  MoveL 769 to (-578.4, 1200, 50) mm, rotated rx -180 ry 0 rz 90 deg; joints [-4.57, -97.989, 142.035, 22.266, 7.604, -25.643]
  MoveL 770 to (-578.4, 1200, -0.5) mm, rotated rx -180 ry 0 rz 90 deg; joints [-4.57, -94.77, 142.936, 44.544, 4.099, -48.025]
  MoveL 771 to (-578.4, 1200, 50) mm, rotated rx -180 ry 0 rz 90 deg; joints [-4.57, -97.989, 142.035, 22.266, 7.604, -25.643]
  MoveL 772 to (-578.4, 1250, 50) mm, rotated rx -180 ry 0 rz 90 deg; joints [-4.804, -101.028, 144.386, 21.399, 8.305, -24.931]
  MoveL 773 to (-578.4, 1250, -0.5) mm, rotated rx 180 ry 0 rz 90 deg; joints [-4.804, -97.638, 145.343, 41.717, 4.543, -45.364]
  MoveL 774 to (-578.4, 1250, 50) mm, rotated rx -180 ry 0 rz 90 deg; joints [-4.804, -101.028, 144.386, 21.399, 8.305, -24.931]
  MoveL 775 to (-578.4, 1300, 50) mm, rotated rx -180 ry 0 rz 90 deg; joints [-5.063, -104.304, 146.692, 20.148, 9.28, -23.844]
  MoveL 776 to (-578.4, 1300, -0.5) mm, rotated rx 180 ry 0 rz 90 deg; joints [-5.063, -100.735, 147.713, 37.677, 5.214, -41.502]
  MoveL 777 to (-578.4, 1300, 50) mm, rotated rx -180 ry 0 rz 90 deg; joints [-5.063, -104.304, 146.692, 20.148, 9.28, -23.844]
  MoveL 778 to (-578.4, 1350, 50) mm, rotated rx 180 ry 0 rz 90 deg; joints [-5.353, -107.868, 148.948, 18.637, 10.585, -22.506]
  MoveL 779 to (-578.4, 1350, -0.5) mm, rotated rx 180 ry 0 rz 90 deg; joints [-5.353, -104.114, 150.044, 33.013, 6.186, -37.025]
  MoveL 780 to (-578.4, 1350, 50) mm, rotated rx 180 ry 0 rz 90 deg; joints [-5.353, -107.868, 148.948, 18.637, 10.585, -22.506]
  MoveL 781 to (-578.4, 1400, 50) mm, rotated rx 180 ry 0 rz 90 deg; joints [-5.676, -111.783, 151.148, 16.997, 12.295, -21.046]
  MoveL 782 to (-578.4, 1400, -0.5) mm, rotated rx 180 ry 0 rz 90 deg; joints [-5.676, -107.847, 152.329, 28.286, 7.548, -32.495]
  MoveL 783 to (-578.4, 1400, 50) mm, rotated rx 180 ry 0 rz 90 deg; joints [-5.676, -111.783, 151.148, 16.997, 12.295, -21.046]
  MoveL 784 to (-578.4, 1450, 50) mm, rotated rx -180 ry 0 rz 90 deg; joints [-6.042, -116.128, 153.28, 15.341, 14.499, -19.577]
  MoveL 785 to (-578.4, 1450, -0.5) mm, rotated rx 180 ry 0 rz 90 deg; joints [-6.042, -112.023, 154.561, 23.895, 9.412, -28.311]
  MoveL 786 to (-578.4, 1450, 50) mm, rotated rx -180 ry 0 rz 90 deg; joints [-6.042, -116.128, 153.28, 15.341, 14.499, -19.577]
  MoveL 787 to (-514.2, 300, 50) mm, rotated rx 180 ry 0 rz 90 deg; joints [-4.34, -58.339, 92.264, 9.183, 17.364, -12.147]
  MoveL 788 to (-514.2, 300, -0.5) mm, rotated rx -180 ry 0 rz 90 deg; joints [-4.34, -56.823, 92.789, 10.363, 15.353, -13.377]
  MoveL 789 to (-514.2, 300, 50) mm, rotated rx 180 ry 0 rz 90 deg; joints [-4.34, -58.339, 92.264, 9.183, 17.364, -12.147]
  MoveL 790 to (-514.2, 650, 50) mm, rotated rx -180 ry 0 rz 90 deg; joints [-5.302, -72.243, 113.368, 18.554, 10.531, -22.388]
  MoveL 791 to (-514.2, 650, -0.5) mm, rotated rx 180 ry 0 rz 90 deg; joints [-5.302, -70.292, 113.949, 24.154, 8.171, -28.062]
  MoveL 792 to (-514.2, 650, 50) mm, rotated rx -180 ry 0 rz 90 deg; joints [-5.302, -72.243, 113.368, 18.554, 10.531, -22.388]
  MoveL 793 to (-476, 230, 50) mm, rotated rx -180 ry 0 rz 90 deg; joints [-5.28, -55.357, 87.377, 10.054, 19.374, -13.603]
  MoveL 794 to (-476, 230, -0.5) mm, rotated rx 180 ry 0 rz 90 deg; joints [-5.28, -53.915, 87.901, 11.14, 17.442, -14.748]
  MoveL 795 to (-476, 230, 50) mm, rotated rx -180 ry 0 rz 90 deg; joints [-5.28, -55.357, 87.377, 10.054, 19.374, -13.603]
  MoveL 796 to (-514.2, 230, 50) mm, rotated rx 180 ry 0 rz 90 deg; joints [-4.188, -55.487, 87.593, 8.057, 19.144, -10.874]
  MoveL 797 to (-514.2, 230, -0.5) mm, rotated rx -180 ry 0 rz 90 deg; joints [-4.188, -54.042, 88.116, 8.943, 17.198, -11.807]
  MoveL 798 to (-514.2, 230, 50) mm, rotated rx 180 ry 0 rz 90 deg; joints [-4.188, -55.487, 87.593, 8.057, 19.144, -10.874]
  MoveL 799 to (-552.4, 230, 50) mm, rotated rx -180 ry 0 rz 90 deg; joints [-3.094, -55.587, 87.758, 5.998, 18.966, -8.08]
  MoveL 800 to (-552.4, 230, -0.5) mm, rotated rx -180 ry 0 rz 90 deg; joints [-3.094, -54.14, 88.282, 6.668, 17.007, -8.784]
  MoveL 801 to (-552.4, 230, 50) mm, rotated rx -180 ry 0 rz 90 deg; joints [-3.094, -55.587, 87.758, 5.998, 18.966, -8.08]
  MoveL 802 to (-655, 50, 50) mm, rotated rx 180 ry 0 rz 90 deg; joints [-0.132, -48.006, 74.913, 0.203, 24.093, -0.288]
  MoveL 803 to (-655, 50, -0.5) mm, rotated rx 180 ry 0 rz 90 deg; joints [-0.132, -46.724, 75.45, 0.219, 22.275, -0.305]
  MoveL 804 to (-655, 50, 50) mm, rotated rx 180 ry 0 rz 90 deg; joints [-0.132, -48.006, 74.913, 0.203, 24.093, -0.288]
  MoveL 805 to (-655, 100, 50) mm, rotated rx 180 ry 0 rz 90 deg; joints [-0.135, -50.213, 78.713, 0.222, 22.501, -0.31]
  MoveL 806 to (-655, 100, -0.5) mm, rotated rx 180 ry 0 rz 90 deg; joints [-0.135, -48.886, 79.243, 0.241, 20.644, -0.331]
  MoveL 807 to (-655, 100, 50) mm, rotated rx 180 ry 0 rz 90 deg; joints [-0.135, -50.213, 78.713, 0.222, 22.501, -0.31]
  MoveL 808 to (-655, 150, 50) mm, rotated rx 180 ry 0 rz 90 deg; joints [-0.138, -52.362, 82.367, 0.243, 20.996, -0.334]
  MoveL 809 to (-655, 150, -0.5) mm, rotated rx -180 ry 0 rz 90 deg; joints [-0.138, -50.989, 82.893, 0.266, 19.097, -0.359]
  MoveL 810 to (-655, 150, 50) mm, rotated rx 180 ry 0 rz 90 deg; joints [-0.138, -52.362, 82.367, 0.243, 20.996, -0.334]
  MoveL 811 to (-655, 200, 50) mm, rotated rx 180 ry 0 rz 90 deg; joints [-0.142, -54.464, 85.894, 0.266, 19.57, -0.361]
  MoveL 812 to (-655, 200, -0.5) mm, rotated rx 180 ry 0 rz 90 deg; joints [-0.142, -53.043, 86.418, 0.295, 17.626, -0.391]
  MoveL 813 to (-655, 200, 50) mm, rotated rx 180 ry 0 rz 90 deg; joints [-0.142, -54.464, 85.894, 0.266, 19.57, -0.361]
  MoveL 814 to (-655, 250, 50) mm, rotated rx 180 ry 0 rz 90 deg; joints [-0.145, -56.528, 89.31, 0.293, 18.219, -0.391]
  MoveL 815 to (-655, 250, -0.5) mm, rotated rx 180 ry 0 rz 90 deg; joints [-0.145, -55.058, 89.833, 0.327, 16.225, -0.427]
  MoveL 816 to (-655, 250, 50) mm, rotated rx 180 ry 0 rz 90 deg; joints [-0.145, -56.528, 89.31, 0.293, 18.219, -0.391]
  MoveL 817 to (-655, 300, 50) mm, rotated rx -180 ry 0 rz 90 deg; joints [-0.149, -58.562, 92.626, 0.322, 16.937, -0.424]
  MoveL 818 to (-655, 300, -0.5) mm, rotated rx 180 ry 0 rz 90 deg; joints [-0.149, -57.041, 93.151, 0.365, 14.89, -0.469]
  MoveL 819 to (-655, 300, 50) mm, rotated rx -180 ry 0 rz 90 deg; joints [-0.149, -58.562, 92.626, 0.322, 16.937, -0.424]
  MoveL 820 to (-655, 350, 50) mm, rotated rx 180 ry 0 rz 90 deg; joints [-0.153, -60.573, 95.852, 0.356, 15.721, -0.461]
  MoveL 821 to (-655, 350, -0.5) mm, rotated rx -180 ry 0 rz 90 deg; joints [-0.153, -58.998, 96.381, 0.409, 13.618, -0.517]
  MoveL 822 to (-655, 350, 50) mm, rotated rx 180 ry 0 rz 90 deg; joints [-0.153, -60.573, 95.852, 0.356, 15.721, -0.461]
  MoveL 823 to (-655, 400, 50) mm, rotated rx -180 ry 0 rz 90 deg; joints [-0.157, -62.568, 98.998, 0.394, 14.57, -0.503]
  MoveL 824 to (-655, 400, -0.5) mm, rotated rx 180 ry 0 rz 90 deg; joints [-0.157, -60.937, 99.532, 0.461, 12.406, -0.572]
  MoveL 825 to (-655, 400, 50) mm, rotated rx -180 ry 0 rz 90 deg; joints [-0.157, -62.568, 98.998, 0.394, 14.57, -0.503]
  MoveL 826 to (-655, 450, 50) mm, rotated rx -180 ry 0 rz 90 deg; joints [-0.162, -64.553, 102.071, 0.437, 13.482, -0.55]
  MoveL 827 to (-655, 450, -0.5) mm, rotated rx 180 ry 0 rz 90 deg; joints [-0.162, -62.863, 102.612, 0.522, 11.252, -0.637]
  MoveL 828 to (-655, 450, 50) mm, rotated rx -180 ry 0 rz 90 deg; joints [-0.162, -64.553, 102.071, 0.437, 13.482, -0.55]
  MoveL 829 to (-655, 500, 50) mm, rotated rx -180 ry 0 rz 90 deg; joints [-0.166, -66.534, 105.078, 0.486, 12.457, -0.604]
  MoveL 830 to (-655, 500, -0.5) mm, rotated rx -180 ry 0 rz 90 deg; joints [-0.166, -64.782, 105.626, 0.594, 10.157, -0.714]
  MoveL 831 to (-655, 500, 50) mm, rotated rx -180 ry 0 rz 90 deg; joints [-0.166, -66.534, 105.078, 0.486, 12.457, -0.604]
  MoveL 832 to (-655, 550, 50) mm, rotated rx 180 ry 0 rz 90 deg; joints [-0.171, -68.517, 108.023, 0.541, 11.495, -0.664]
  MoveL 833 to (-655, 550, -0.5) mm, rotated rx -180 ry 0 rz 90 deg; joints [-0.171, -66.7, 108.581, 0.681, 9.12, -0.805]
  MoveL 834 to (-655, 550, 50) mm, rotated rx 180 ry 0 rz 90 deg; joints [-0.171, -68.517, 108.023, 0.541, 11.495, -0.664]
  MoveL 835 to (-655, 600, 50) mm, rotated rx -180 ry 0 rz 90 deg; joints [-0.177, -70.508, 110.911, 0.605, 10.598, -0.732]
  MoveL 836 to (-655, 600, -0.5) mm, rotated rx -180 ry 0 rz 90 deg; joints [-0.177, -68.622, 111.481, 0.785, 8.142, -0.915]
  MoveL 837 to (-655, 600, 50) mm, rotated rx -180 ry 0 rz 90 deg; joints [-0.177, -70.508, 110.911, 0.605, 10.598, -0.732]
  MoveL 838 to (-655, 650, 50) mm, rotated rx -180 ry 0 rz 90 deg; joints [-0.182, -72.515, 113.748, 0.676, 9.768, -0.808]
  MoveL 839 to (-655, 650, -0.5) mm, rotated rx 180 ry 0 rz 90 deg; joints [-0.182, -70.554, 114.33, 0.913, 7.225, -1.047]
  MoveL 840 to (-655, 650, 50) mm, rotated rx -180 ry 0 rz 90 deg; joints [-0.182, -72.515, 113.748, 0.676, 9.768, -0.808]
  MoveL 841 to (-655, 700, 50) mm, rotated rx 180 ry 0 rz 90 deg; joints [-0.188, -74.542, 116.535, 0.757, 9.008, -0.894]
  MoveL 842 to (-655, 700, -0.5) mm, rotated rx 180 ry 0 rz 90 deg; joints [-0.188, -72.503, 117.133, 1.068, 6.371, -1.208]
  MoveL 843 to (-655, 700, 50) mm, rotated rx 180 ry 0 rz 90 deg; joints [-0.188, -74.542, 116.535, 0.757, 9.008, -0.894]
  MoveL 844 to (-655, 750, 50) mm, rotated rx -180 ry 0 rz 90 deg; joints [-0.195, -76.598, 119.277, 0.847, 8.323, -0.989]
  MoveL 845 to (-655, 750, -0.5) mm, rotated rx 180 ry 0 rz 90 deg; joints [-0.195, -74.475, 119.891, 1.26, 5.585, -1.405]
  MoveL 846 to (-655, 750, 50) mm, rotated rx -180 ry 0 rz 90 deg; joints [-0.195, -76.598, 119.277, 0.847, 8.323, -0.989]
  MoveL 847 to (-655, 800, 50) mm, rotated rx -180 ry 0 rz 90 deg; joints [-0.202, -78.691, 121.976, 0.945, 7.717, -1.093]
  MoveL 848 to (-655, 800, -0.5) mm, rotated rx 180 ry 0 rz 90 deg; joints [-0.202, -76.477, 122.609, 1.495, 4.87, -1.646]
  MoveL 849 to (-655, 800, 50) mm, rotated rx -180 ry 0 rz 90 deg; joints [-0.202, -78.691, 121.976, 0.945, 7.717, -1.093]
  MoveL 850 to (-655, 850, 50) mm, rotated rx 180 ry 0 rz 90 deg; joints [-0.209, -80.83, 124.634, 1.05, 7.198, -1.204]
  MoveL 851 to (-655, 850, -0.5) mm, rotated rx -180 ry 0 rz 90 deg; joints [-0.209, -78.519, 125.288, 1.782, 4.233, -1.94]
  MoveL 852 to (-655, 850, 50) mm, rotated rx 180 ry 0 rz 90 deg; joints [-0.209, -80.83, 124.634, 1.05, 7.198, -1.204]
  MoveL 853 to (-655, 900, 50) mm, rotated rx 180 ry 0 rz 90 deg; joints [-0.217, -83.024, 127.252, 1.157, 6.773, -1.318]
  MoveL 854 to (-655, 900, -0.5) mm, rotated rx -180 ry 0 rz 90 deg; joints [-0.217, -80.609, 127.931, 2.127, 3.681, -2.291]
  MoveL 855 to (-655, 900, 50) mm, rotated rx 180 ry 0 rz 90 deg; joints [-0.217, -83.024, 127.252, 1.157, 6.773, -1.318]
  MoveL 856 to (-655, 950, 50) mm, rotated rx 180 ry 0 rz 90 deg; joints [-0.225, -85.286, 129.834, 1.262, 6.454, -1.429]
  MoveL 857 to (-655, 950, -0.5) mm, rotated rx 180 ry 0 rz 90 deg; joints [-0.225, -82.759, 130.54, 2.524, 3.223, -2.695]
  MoveL 858 to (-655, 950, 50) mm, rotated rx 180 ry 0 rz 90 deg; joints [-0.225, -85.286, 129.834, 1.262, 6.454, -1.429]
  MoveL 859 to (-655, 1000, 50) mm, rotated rx 180 ry 0 rz 90 deg; joints [-0.235, -87.628, 132.378, 1.356, 6.252, -1.53]
  MoveL 860 to (-655, 1000, -0.5) mm, rotated rx 180 ry 0 rz 90 deg; joints [-0.235, -84.981, 133.115, 2.95, 2.87, -3.129]
  MoveL 861 to (-655, 1000, 50) mm, rotated rx 180 ry 0 rz 90 deg; joints [-0.235, -87.628, 132.378, 1.356, 6.252, -1.53]
  MoveL 862 to (-655, 1050, 50) mm, rotated rx 180 ry 0 rz 90 deg; joints [-0.245, -90.068, 134.886, 1.429, 6.184, -1.611]
  MoveL 863 to (-655, 1050, -0.5) mm, rotated rx 180 ry 0 rz 90 deg; joints [-0.245, -87.291, 135.657, 3.347, 2.638, -3.534]
  MoveL 864 to (-655, 1050, 50) mm, rotated rx 180 ry 0 rz 90 deg; joints [-0.245, -90.068, 134.886, 1.429, 6.184, -1.611]
  MoveL 865 to (-655, 1100, 50) mm, rotated rx 180 ry 0 rz 90 deg; joints [-0.256, -92.624, 137.358, 1.473, 6.268, -1.663]
  MoveL 866 to (-655, 1100, -0.5) mm, rotated rx -180 ry 0 rz 90 deg; joints [-0.256, -89.706, 138.168, 3.626, 2.544, -3.821]
  MoveL 867 to (-655, 1100, 50) mm, rotated rx 180 ry 0 rz 90 deg; joints [-0.256, -92.624, 137.358, 1.473, 6.268, -1.663]
  MoveL 868 to (-655, 1150, 50) mm, rotated rx -180 ry 0 rz 90 deg; joints [-0.267, -95.319, 139.793, 1.481, 6.528, -1.679]
  MoveL 869 to (-655, 1150, -0.5) mm, rotated rx -180 ry 0 rz 90 deg; joints [-0.267, -92.25, 140.647, 3.7, 2.609, -3.904]
  MoveL 870 to (-655, 1150, 50) mm, rotated rx -180 ry 0 rz 90 deg; joints [-0.267, -95.319, 139.793, 1.481, 6.528, -1.679]
  MoveL 871 to (-655, 1200, 50) mm, rotated rx -180 ry 0 rz 90 deg; joints [-0.281, -98.18, 142.19, 1.45, 6.993, -1.658]
  MoveL 872 to (-655, 1200, -0.5) mm, rotated rx 180 ry 0 rz 90 deg; joints [-0.281, -94.951, 143.093, 3.537, 2.863, -3.751]
  MoveL 873 to (-655, 1200, 50) mm, rotated rx -180 ry 0 rz 90 deg; joints [-0.281, -98.18, 142.19, 1.45, 6.993, -1.658]
  MoveL 874 to (-655, 1250, 50) mm, rotated rx 180 ry 0 rz 90 deg; joints [-0.295, -101.244, 144.545, 1.386, 7.701, -1.603]
  MoveL 875 to (-655, 1250, -0.5) mm, rotated rx 180 ry 0 rz 90 deg; joints [-0.295, -97.842, 145.506, 3.187, 3.342, -3.411]
  MoveL 876 to (-655, 1250, 50) mm, rotated rx 180 ry 0 rz 90 deg; joints [-0.295, -101.244, 144.545, 1.386, 7.701, -1.603]
  MoveL 877 to (-783.4, 50, 50) mm, rotated rx 180 ry 0 rz 90 deg; joints [3.253, -47.849, 74.641, -4.972, 24.334, 7.062]
  MoveL 878 to (-783.4, 50, -0.5) mm, rotated rx 180 ry 0 rz 90 deg; joints [3.253, -46.571, 75.179, -5.349, 22.525, 7.473]
  MoveL 879 to (-783.4, 50, 50) mm, rotated rx 180 ry 0 rz 90 deg; joints [3.253, -47.849, 74.641, -4.972, 24.334, 7.062]
  MoveL 880 to (-783.4, 100, 50) mm, rotated rx 180 ry 0 rz 90 deg; joints [3.33, -50.057, 78.445, -5.424, 22.75, 7.593]
  MoveL 881 to (-783.4, 100, -0.5) mm, rotated rx -180 ry 0 rz 90 deg; joints [3.33, -48.733, 78.976, -5.88, 20.905, 8.084]
  MoveL 882 to (-783.4, 100, 50) mm, rotated rx 180 ry 0 rz 90 deg; joints [3.33, -50.057, 78.445, -5.424, 22.75, 7.593]
  MoveL 883 to (-783.4, 150, 50) mm, rotated rx 180 ry 0 rz 90 deg; joints [3.41, -52.206, 82.103, -5.926, 21.256, 8.177]
  MoveL 884 to (-783.4, 150, -0.5) mm, rotated rx 180 ry 0 rz 90 deg; joints [3.41, -50.837, 82.629, -6.48, 19.371, 8.767]
  MoveL 885 to (-783.4, 150, 50) mm, rotated rx 180 ry 0 rz 90 deg; joints [3.41, -52.206, 82.103, -5.926, 21.256, 8.177]
  MoveL 886 to (-783.4, 200, 50) mm, rotated rx -180 ry 0 rz 90 deg; joints [3.494, -54.308, 85.633, -6.488, 19.844, 8.822]
  MoveL 887 to (-783.4, 200, -0.5) mm, rotated rx -180 ry 0 rz 90 deg; joints [3.494, -52.89, 86.157, -7.162, 17.917, 9.535]
  MoveL 888 to (-783.4, 200, 50) mm, rotated rx -180 ry 0 rz 90 deg; joints [3.494, -54.308, 85.633, -6.488, 19.844, 8.822]
  MoveL 889 to (-783.4, 250, 50) mm, rotated rx 180 ry 0 rz 90 deg; joints [3.583, -56.37, 89.05, -7.116, 18.508, 9.537]
  MoveL 890 to (-783.4, 250, -0.5) mm, rotated rx -180 ry 0 rz 90 deg; joints [3.583, -54.904, 89.574, -7.942, 16.535, 10.403]
  MoveL 891 to (-783.4, 250, 50) mm, rotated rx 180 ry 0 rz 90 deg; joints [3.583, -56.37, 89.05, -7.116, 18.508, 9.537]
  MoveL 892 to (-783.4, 300, 50) mm, rotated rx 180 ry 0 rz 90 deg; joints [3.676, -58.402, 92.367, -7.822, 17.244, 10.332]
  MoveL 893 to (-783.4, 300, -0.5) mm, rotated rx -180 ry 0 rz 90 deg; joints [3.676, -56.885, 92.892, -8.838, 15.223, 11.391]
  MoveL 894 to (-783.4, 300, 50) mm, rotated rx 180 ry 0 rz 90 deg; joints [3.676, -58.402, 92.367, -7.822, 17.244, 10.332]
  MoveL 895 to (-783.4, 350, 50) mm, rotated rx 180 ry 0 rz 90 deg; joints [3.774, -60.41, 95.593, -8.616, 16.05, 11.219]
  MoveL 896 to (-783.4, 350, -0.5) mm, rotated rx 180 ry 0 rz 90 deg; joints [3.774, -58.84, 96.122, -9.873, 13.978, 12.52]
  MoveL 897 to (-783.4, 350, 50) mm, rotated rx 180 ry 0 rz 90 deg; joints [3.774, -60.41, 95.593, -8.616, 16.05, 11.219]
  MoveL 898 to (-783.4, 400, 50) mm, rotated rx 180 ry 0 rz 90 deg; joints [3.877, -62.402, 98.739, -9.51, 14.923, 12.21]
  MoveL 899 to (-783.4, 400, -0.5) mm, rotated rx 180 ry 0 rz 90 deg; joints [3.877, -60.776, 99.272, -11.074, 12.799, 13.82]
  MoveL 900 to (-783.4, 400, 50) mm, rotated rx 180 ry 0 rz 90 deg; joints [3.877, -62.402, 98.739, -9.51, 14.923, 12.21]
  MoveL 901 to (-783.4, 450, 50) mm, rotated rx 180 ry 0 rz 90 deg; joints [3.986, -64.383, 101.811, -10.519, 13.864, 13.319]
  MoveL 902 to (-783.4, 450, -0.5) mm, rotated rx 180 ry 0 rz 90 deg; joints [3.986, -62.698, 102.35, -12.474, 11.685, 15.323]
  MoveL 903 to (-783.4, 450, 50) mm, rotated rx 180 ry 0 rz 90 deg; joints [3.986, -64.383, 101.811, -10.519, 13.864, 13.319]
  MoveL 904 to (-783.4, 500, 50) mm, rotated rx -180 ry 0 rz 90 deg; joints [4.101, -66.359, 104.815, -11.656, 12.873, 14.56]
  MoveL 905 to (-783.4, 500, -0.5) mm, rotated rx -180 ry 0 rz 90 deg; joints [4.101, -64.613, 105.363, -14.114, 10.636, 17.071]
  MoveL 906 to (-783.4, 500, 50) mm, rotated rx -180 ry 0 rz 90 deg; joints [4.101, -66.359, 104.815, -11.656, 12.873, 14.56]
  MoveL 907 to (-783.4, 550, 50) mm, rotated rx 180 ry 0 rz 90 deg; joints [4.224, -68.337, 107.758, -12.935, 11.95, 15.949]
  MoveL 908 to (-783.4, 550, -0.5) mm, rotated rx 180 ry 0 rz 90 deg; joints [4.224, -66.525, 108.315, -16.041, 9.656, 19.11]
  MoveL 909 to (-783.4, 550, 50) mm, rotated rx 180 ry 0 rz 90 deg; joints [4.224, -68.337, 107.758, -12.935, 11.95, 15.949]
  MoveL 910 to (-783.4, 600, 50) mm, rotated rx 180 ry 0 rz 90 deg; joints [4.353, -70.321, 110.643, -14.369, 11.098, 17.497]
  MoveL 911 to (-783.4, 600, -0.5) mm, rotated rx 180 ry 0 rz 90 deg; joints [4.353, -68.441, 111.211, -18.308, 8.747, 21.495]
  MoveL 912 to (-783.4, 600, 50) mm, rotated rx 180 ry 0 rz 90 deg; joints [4.353, -70.321, 110.643, -14.369, 11.098, 17.497]
  MoveL 913 to (-783.4, 650, 50) mm, rotated rx -180 ry 0 rz 90 deg; joints [4.491, -72.32, 113.476, -15.967, 10.32, 19.215]
  MoveL 914 to (-783.4, 650, -0.5) mm, rotated rx 180 ry 0 rz 90 deg; joints [4.491, -70.367, 114.057, -20.973, 7.914, 24.283]
  MoveL 915 to (-783.4, 650, 50) mm, rotated rx -180 ry 0 rz 90 deg; joints [4.491, -72.32, 113.476, -15.967, 10.32, 19.215]
  MoveL 916 to (-783.4, 700, 50) mm, rotated rx 180 ry 0 rz 90 deg; joints [4.638, -74.339, 116.259, -17.729, 9.621, 21.103]
  MoveL 917 to (-783.4, 700, -0.5) mm, rotated rx -180 ry 0 rz 90 deg; joints [4.638, -72.307, 116.855, -24.09, 7.162, 27.531]
  MoveL 918 to (-783.4, 700, 50) mm, rotated rx 180 ry 0 rz 90 deg; joints [4.638, -74.339, 116.259, -17.729, 9.621, 21.103]
  MoveL 919 to (-783.4, 750, 50) mm, rotated rx -180 ry 0 rz 90 deg; joints [4.795, -76.385, 118.996, -19.645, 9.003, 23.152]
  MoveL 920 to (-783.4, 750, -0.5) mm, rotated rx 180 ry 0 rz 90 deg; joints [4.795, -74.27, 119.609, -27.698, 6.499, 31.277]
  MoveL 921 to (-783.4, 750, 50) mm, rotated rx -180 ry 0 rz 90 deg; joints [4.795, -76.385, 118.996, -19.645, 9.003, 23.152]
  MoveL 922 to (-783.4, 800, 50) mm, rotated rx 180 ry 0 rz 90 deg; joints [4.963, -78.466, 121.689, -21.685, 8.473, 25.331]
  MoveL 923 to (-783.4, 800, -0.5) mm, rotated rx -180 ry 0 rz 90 deg; joints [4.963, -76.262, 122.321, -31.796, 5.931, 35.519]
  MoveL 924 to (-783.4, 800, 50) mm, rotated rx 180 ry 0 rz 90 deg; joints [4.963, -78.466, 121.689, -21.685, 8.473, 25.331]
  MoveL 925 to (-783.4, 850, 50) mm, rotated rx -180 ry 0 rz 90 deg; joints [5.143, -80.591, 124.341, -23.797, 8.038, 27.59]
  MoveL 926 to (-783.4, 850, -0.5) mm, rotated rx -180 ry 0 rz 90 deg; joints [5.143, -78.291, 124.994, -36.311, 5.467, 40.188]
  MoveL 927 to (-783.4, 850, 50) mm, rotated rx -180 ry 0 rz 90 deg; joints [5.143, -80.591, 124.341, -23.797, 8.038, 27.59]
  MoveL 928 to (-783.4, 900, 50) mm, rotated rx 180 ry 0 rz 90 deg; joints [5.337, -82.769, 126.954, -25.896, 7.702, 29.845]
  MoveL 929 to (-783.4, 900, -0.5) mm, rotated rx 180 ry 0 rz 90 deg; joints [5.337, -80.366, 127.63, -41.068, 5.112, 45.108]
  MoveL 930 to (-783.4, 900, 50) mm, rotated rx 180 ry 0 rz 90 deg; joints [5.337, -82.769, 126.954, -25.896, 7.702, 29.845]
  MoveL 931 to (-783.4, 950, 50) mm, rotated rx -180 ry 0 rz 90 deg; joints [5.546, -85.012, 129.528, -27.873, 7.475, 31.986]
  MoveL 932 to (-783.4, 950, -0.5) mm, rotated rx 180 ry 0 rz 90 deg; joints [5.546, -82.499, 130.23, -45.773, 4.869, 49.985]
  MoveL 933 to (-783.4, 950, 50) mm, rotated rx -180 ry 0 rz 90 deg; joints [5.546, -85.012, 129.528, -27.873, 7.475, 31.986]
  MoveL 934 to (-783.4, 1000, 50) mm, rotated rx -180 ry 0 rz 90 deg; joints [5.771, -87.332, 132.064, -29.593, 7.362, 33.881]
  MoveL 935 to (-783.4, 1000, -0.5) mm, rotated rx 180 ry 0 rz 90 deg; joints [5.771, -84.701, 132.797, -50.034, 4.736, 54.429]
  MoveL 936 to (-783.4, 1000, 50) mm, rotated rx -180 ry 0 rz 90 deg; joints [5.771, -87.332, 132.064, -29.593, 7.362, 33.881]
  MoveL 937 to (-783.4, 1050, 50) mm, rotated rx -180 ry 0 rz 90 deg; joints [6.016, -89.746, 134.564, -30.915, 7.376, 35.388]
  MoveL 938 to (-783.4, 1050, -0.5) mm, rotated rx -180 ry 0 rz 90 deg; joints [6.016, -86.986, 135.33, -53.428, 4.711, 58.018]
  MoveL 939 to (-783.4, 1050, 50) mm, rotated rx -180 ry 0 rz 90 deg; joints [6.016, -89.746, 134.564, -30.915, 7.376, 35.388]
  MoveL 940 to (-783.4, 1100, 50) mm, rotated rx 180 ry 0 rz 90 deg; joints [6.282, -92.271, 137.026, -31.715, 7.527, 36.384]
  MoveL 941 to (-783.4, 1100, -0.5) mm, rotated rx 180 ry 0 rz 90 deg; joints [6.282, -89.373, 137.83, -55.58, 4.789, 60.376]
  MoveL 942 to (-783.4, 1100, 50) mm, rotated rx 180 ry 0 rz 90 deg; joints [6.282, -92.271, 137.026, -31.715, 7.527, 36.384]
  MoveL 943 to (-783.4, 1150, 50) mm, rotated rx 180 ry 0 rz 90 deg; joints [6.573, -94.928, 139.451, -31.906, 7.834, 36.783]
  MoveL 944 to (-783.4, 1150, -0.5) mm, rotated rx 180 ry 0 rz 90 deg; joints [6.573, -91.882, 140.298, -56.229, 4.971, 61.246]
  MoveL 945 to (-783.4, 1150, 50) mm, rotated rx 180 ry 0 rz 90 deg; joints [6.573, -94.928, 139.451, -31.906, 7.834, 36.783]
  MoveL 946 to (-783.4, 1200, 50) mm, rotated rx -180 ry 0 rz 90 deg; joints [6.892, -97.744, 141.837, -31.458, 8.32, 36.555]
  MoveL 947 to (-783.4, 1200, -0.5) mm, rotated rx 180 ry 0 rz 90 deg; joints [6.892, -94.539, 142.732, -55.267, 5.272, 60.519]
  MoveL 948 to (-783.4, 1200, 50) mm, rotated rx -180 ry 0 rz 90 deg; joints [6.892, -97.744, 141.837, -31.458, 8.32, 36.555]
  MoveL 949 to (-783.4, 1250, 50) mm, rotated rx -180 ry 0 rz 90 deg; joints [7.243, -100.751, 144.181, -30.408, 9.019, 35.739]
  MoveL 950 to (-783.4, 1250, -0.5) mm, rotated rx -180 ry 0 rz 90 deg; joints [7.243, -97.377, 145.132, -52.756, 5.72, 58.259]
  MoveL 951 to (-783.4, 1250, 50) mm, rotated rx -180 ry 0 rz 90 deg; joints [7.243, -100.751, 144.181, -30.408, 9.019, 35.739]
  MoveL 952 to (-719.2, 300, 50) mm, rotated rx -180 ry 0 rz 90 deg; joints [1.765, -58.525, 92.566, -3.8, 17.007, 5.006]
  MoveL 953 to (-719.2, 300, -0.5) mm, rotated rx 180 ry 0 rz 90 deg; joints [1.765, -57.005, 93.092, -4.305, 14.967, 5.531]
  MoveL 954 to (-719.2, 300, 50) mm, rotated rx -180 ry 0 rz 90 deg; joints [1.765, -58.525, 92.566, -3.8, 17.007, 5.006]
  MoveL 955 to (-719.2, 650, 50) mm, rotated rx -180 ry 0 rz 90 deg; joints [2.158, -72.47, 113.685, -7.925, 9.897, 9.486]
  MoveL 956 to (-719.2, 650, -0.5) mm, rotated rx -180 ry 0 rz 90 deg; joints [2.158, -70.511, 114.268, -10.62, 7.389, 12.211]
  MoveL 957 to (-719.2, 650, 50) mm, rotated rx -180 ry 0 rz 90 deg; joints [2.158, -72.47, 113.685, -7.925, 9.897, 9.486]
  MoveL 958 to (-681, 230, 50) mm, rotated rx 180 ry 0 rz 90 deg; joints [0.604, -55.702, 87.949, -1.183, 18.759, 1.59]
  MoveL 959 to (-681, 230, -0.5) mm, rotated rx 180 ry 0 rz 90 deg; joints [0.604, -54.252, 88.472, -1.317, 16.785, 1.731]
  MoveL 960 to (-681, 230, 50) mm, rotated rx 180 ry 0 rz 90 deg; joints [0.604, -55.702, 87.949, -1.183, 18.759, 1.59]
  MoveL 961 to (-719.2, 230, 50) mm, rotated rx 180 ry 0 rz 90 deg; joints [1.703, -55.671, 87.897, -3.325, 18.816, 4.471]
  MoveL 962 to (-719.2, 230, -0.5) mm, rotated rx 180 ry 0 rz 90 deg; joints [1.703, -54.221, 88.42, -3.7, 16.847, 4.866]
  MoveL 963 to (-719.2, 230, 50) mm, rotated rx 180 ry 0 rz 90 deg; joints [1.703, -55.671, 87.897, -3.325, 18.816, 4.471]
  MoveL 964 to (-757.4, 230, 50) mm, rotated rx 180 ry 0 rz 90 deg; joints [2.801, -55.609, 87.794, -5.44, 18.927, 7.325]
  MoveL 965 to (-757.4, 230, -0.5) mm, rotated rx 180 ry 0 rz 90 deg; joints [2.801, -54.161, 88.318, -6.049, 16.966, 7.965]
  MoveL 966 to (-757.4, 230, 50) mm, rotated rx 180 ry 0 rz 90 deg; joints [2.801, -55.609, 87.794, -5.44, 18.927, 7.325]
  MoveL 967 to (-681, 420, 50) mm, rotated rx 180 ry 0 rz 90 deg; joints [0.668, -63.358, 100.229, -1.722, 14.137, 2.189]
  MoveL 968 to (-681, 420, -0.5) mm, rotated rx 180 ry 0 rz 90 deg; joints [0.668, -61.704, 100.765, -2.031, 11.949, 2.506]
  MoveL 969 to (-681, 420, 50) mm, rotated rx 180 ry 0 rz 90 deg; joints [0.668, -63.358, 100.229, -1.722, 14.137, 2.189]
  MoveL 970 to (-719.2, 420, 50) mm, rotated rx 180 ry 0 rz 90 deg; joints [1.883, -63.324, 100.176, -4.831, 14.211, 6.147]
  MoveL 971 to (-719.2, 420, -0.5) mm, rotated rx 180 ry 0 rz 90 deg; joints [1.883, -61.672, 100.713, -5.692, 12.032, 7.031]
  MoveL 972 to (-719.2, 420, 50) mm, rotated rx 180 ry 0 rz 90 deg; joints [1.883, -63.324, 100.176, -4.831, 14.211, 6.147]
  MoveL 973 to (-757.4, 420, 50) mm, rotated rx 180 ry 0 rz 90 deg; joints [3.096, -63.258, 100.074, -7.879, 14.355, 10.043]
  MoveL 974 to (-757.4, 420, -0.5) mm, rotated rx 180 ry 0 rz 90 deg; joints [3.096, -61.608, 100.61, -9.26, 12.193, 11.461]
  MoveL 975 to (-757.4, 420, 50) mm, rotated rx 180 ry 0 rz 90 deg; joints [3.096, -63.258, 100.074, -7.879, 14.355, 10.043]
  MoveL 976 to (-681, 1020, 50) mm, rotated rx 180 ry 0 rz 90 deg; joints [1.002, -88.583, 133.377, -5.808, 6.242, 6.552]
  MoveL 977 to (-681, 1020, -0.5) mm, rotated rx -180 ry 0 rz 90 deg; joints [1.002, -85.885, 134.127, -12.858, 2.834, 13.622]
  MoveL 978 to (-681, 1020, 50) mm, rotated rx 180 ry 0 rz 90 deg; joints [1.002, -88.583, 133.377, -5.808, 6.242, 6.552]
  MoveL 979 to (-719.2, 1020, 50) mm, rotated rx 180 ry 0 rz 90 deg; joints [2.822, -88.521, 133.313, -15.913, 6.489, 18.01]
  MoveL 980 to (-719.2, 1020, -0.5) mm, rotated rx -180 ry 0 rz 90 deg; joints [2.822, -85.827, 134.062, -32.408, 3.314, 34.558]
  MoveL 981 to (-719.2, 1020, 50) mm, rotated rx 180 ry 0 rz 90 deg; joints [2.822, -88.521, 133.313, -15.913, 6.489, 18.01]
  MoveL 982 to (-757.4, 1020, 50) mm, rotated rx -180 ry 0 rz 90 deg; joints [4.637, -88.401, 133.188, -24.885, 6.944, 28.331]
  MoveL 983 to (-757.4, 1020, -0.5) mm, rotated rx 180 ry 0 rz 90 deg; joints [4.637, -85.713, 133.935, -45.498, 4.09, 49.032]
  MoveL 984 to (-757.4, 1020, 50) mm, rotated rx -180 ry 0 rz 90 deg; joints [4.637, -88.401, 133.188, -24.885, 6.944, 28.331]
  MoveL 985 to (-890, 50, 50) mm, rotated rx -180 ry 0 rz 90 deg; joints [6.048, -47.46, 73.966, -9.052, 24.924, 12.928]
  MoveL 986 to (-890, 50, -0.5) mm, rotated rx 180 ry 0 rz 90 deg; joints [6.048, -46.189, 74.505, -9.714, 23.138, 13.653]
  MoveL 987 to (-890, 50, 50) mm, rotated rx -180 ry 0 rz 90 deg; joints [6.048, -47.46, 73.966, -9.052, 24.924, 12.928]
  MoveL 988 to (-890, 100, 50) mm, rotated rx -180 ry 0 rz 90 deg; joints [6.189, -49.67, 77.782, -9.853, 23.36, 13.876]
  MoveL 989 to (-890, 100, -0.5) mm, rotated rx 180 ry 0 rz 90 deg; joints [6.189, -48.355, 78.314, -10.648, 21.542, 14.737]
  MoveL 990 to (-890, 100, 50) mm, rotated rx -180 ry 0 rz 90 deg; joints [6.189, -49.67, 77.782, -9.853, 23.36, 13.876]
  MoveL 991 to (-890, 150, 50) mm, rotated rx 180 ry 0 rz 90 deg; joints [6.337, -51.82, 81.449, -10.738, 21.89, 14.913]
  MoveL 992 to (-890, 150, -0.5) mm, rotated rx 180 ry 0 rz 90 deg; joints [6.337, -50.459, 81.976, -11.697, 20.038, 15.939]
  MoveL 993 to (-890, 150, 50) mm, rotated rx 180 ry 0 rz 90 deg; joints [6.337, -51.82, 81.449, -10.738, 21.89, 14.913]
  MoveL 994 to (-890, 200, 50) mm, rotated rx 180 ry 0 rz 90 deg; joints [6.493, -53.92, 84.986, -11.72, 20.508, 16.05]
  MoveL 995 to (-890, 200, -0.5) mm, rotated rx 180 ry 0 rz 90 deg; joints [6.493, -52.512, 85.51, -12.878, 18.619, 17.28]
  MoveL 996 to (-890, 200, 50) mm, rotated rx 180 ry 0 rz 90 deg; joints [6.493, -53.92, 84.986, -11.72, 20.508, 16.05]
  MoveL 997 to (-890, 250, 50) mm, rotated rx -180 ry 0 rz 90 deg; joints [6.656, -55.979, 88.407, -12.811, 19.206, 17.301]
  MoveL 998 to (-890, 250, -0.5) mm, rotated rx 180 ry 0 rz 90 deg; joints [6.656, -54.523, 88.93, -14.215, 17.281, 18.779]
  MoveL 999 to (-890, 250, 50) mm, rotated rx -180 ry 0 rz 90 deg; joints [6.656, -55.979, 88.407, -12.811, 19.206, 17.301]
  MoveL 1000 to (-890, 300, 50) mm, rotated rx -180 ry 0 rz 90 deg; joints [6.828, -58.007, 91.725, -14.024, 17.983, 18.68]
  MoveL 1001 to (-890, 300, -0.5) mm, rotated rx -180 ry 0 rz 90 deg; joints [6.828, -56.5, 92.25, -15.73, 16.02, 20.464]
  MoveL 1002 to (-890, 300, 50) mm, rotated rx -180 ry 0 rz 90 deg; joints [6.828, -58.007, 91.725, -14.024, 17.983, 18.68]
  MoveL 1003 to (-890, 350, 50) mm, rotated rx -180 ry 0 rz 90 deg; joints [7.008, -60.009, 94.952, -15.373, 16.836, 20.201]
  MoveL 1004 to (-890, 350, -0.5) mm, rotated rx 180 ry 0 rz 90 deg; joints [7.008, -58.449, 95.48, -17.453, 14.834, 22.362]
  MoveL 1005 to (-890, 350, 50) mm, rotated rx -180 ry 0 rz 90 deg; joints [7.008, -60.009, 94.952, -15.373, 16.836, 20.201]
  MoveL 1006 to (-890, 400, 50) mm, rotated rx 180 ry 0 rz 90 deg; joints [7.199, -61.992, 98.096, -16.874, 15.764, 21.88]
  MoveL 1007 to (-890, 400, -0.5) mm, rotated rx -180 ry 0 rz 90 deg; joints [7.199, -60.378, 98.628, -19.414, 13.724, 24.506]
  MoveL 1008 to (-890, 400, 50) mm, rotated rx 180 ry 0 rz 90 deg; joints [7.199, -61.992, 98.096, -16.874, 15.764, 21.88]
  MoveL 1009 to (-890, 450, 50) mm, rotated rx 180 ry 0 rz 90 deg; joints [7.4, -63.963, 101.165, -18.54, 14.768, 23.731]
  MoveL 1010 to (-890, 450, -0.5) mm, rotated rx -180 ry 0 rz 90 deg; joints [7.4, -62.292, 101.703, -21.649, 12.692, 26.93]
  MoveL 1011 to (-890, 450, 50) mm, rotated rx 180 ry 0 rz 90 deg; joints [7.4, -63.963, 101.165, -18.54, 14.768, 23.731]
  MoveL 1012 to (-890, 500, 50) mm, rotated rx -180 ry 0 rz 90 deg; joints [7.612, -65.928, 104.165, -20.385, 13.847, 25.769]
  MoveL 1013 to (-890, 500, -0.5) mm, rotated rx 180 ry 0 rz 90 deg; joints [7.612, -64.196, 104.711, -24.19, 11.739, 29.671]
  MoveL 1014 to (-890, 500, 50) mm, rotated rx -180 ry 0 rz 90 deg; joints [7.612, -65.928, 104.165, -20.385, 13.847, 25.769]
  MoveL 1015 to (-890, 550, 50) mm, rotated rx -180 ry 0 rz 90 deg; joints [7.837, -67.892, 107.102, -22.415, 13.006, 28.001]
  MoveL 1016 to (-890, 550, -0.5) mm, rotated rx 180 ry 0 rz 90 deg; joints [7.837, -66.096, 107.656, -27.072, 10.869, 32.759]
  MoveL 1017 to (-890, 550, 50) mm, rotated rx -180 ry 0 rz 90 deg; joints [7.837, -67.892, 107.102, -22.415, 13.006, 28.001]
  MoveL 1018 to (-890, 600, 50) mm, rotated rx 180 ry 0 rz 90 deg; joints [8.076, -69.861, 109.98, -24.635, 12.245, 30.432]
  MoveL 1019 to (-890, 600, -0.5) mm, rotated rx 180 ry 0 rz 90 deg; joints [8.076, -67.997, 110.545, -30.316, 10.087, 36.221]
  MoveL 1020 to (-890, 600, 50) mm, rotated rx 180 ry 0 rz 90 deg; joints [8.076, -69.861, 109.98, -24.635, 12.245, 30.432]
  MoveL 1021 to (-890, 650, 50) mm, rotated rx 180 ry 0 rz 90 deg; joints [8.329, -71.841, 112.804, -27.037, 11.57, 33.055]
  MoveL 1022 to (-890, 650, -0.5) mm, rotated rx 180 ry 0 rz 90 deg; joints [8.329, -69.906, 113.382, -33.932, 9.4, 40.065]
  MoveL 1023 to (-890, 650, 50) mm, rotated rx 180 ry 0 rz 90 deg; joints [8.329, -71.841, 112.804, -27.037, 11.57, 33.055]
  MoveL 1024 to (-890, 700, 50) mm, rotated rx 180 ry 0 rz 90 deg; joints [8.599, -73.838, 115.577, -29.598, 10.983, 35.848]
  MoveL 1025 to (-890, 700, -0.5) mm, rotated rx -180 ry 0 rz 90 deg; joints [8.599, -71.827, 116.169, -37.897, 8.812, 44.271]
  MoveL 1026 to (-890, 700, 50) mm, rotated rx 180 ry 0 rz 90 deg; joints [8.599, -73.838, 115.577, -29.598, 10.983, 35.848]
  MoveL 1027 to (-890, 750, 50) mm, rotated rx -180 ry 0 rz 90 deg; joints [8.887, -75.86, 118.302, -32.281, 10.488, 38.775]
  MoveL 1028 to (-890, 750, -0.5) mm, rotated rx 180 ry 0 rz 90 deg; joints [8.887, -73.767, 118.91, -42.154, 8.329, 48.78]
  MoveL 1029 to (-890, 750, 50) mm, rotated rx -180 ry 0 rz 90 deg; joints [8.887, -75.86, 118.302, -32.281, 10.488, 38.775]
  MoveL 1030 to (-890, 800, 50) mm, rotated rx -180 ry 0 rz 90 deg; joints [9.194, -77.913, 120.983, -35.023, 10.091, 41.774]
  MoveL 1031 to (-890, 800, -0.5) mm, rotated rx 180 ry 0 rz 90 deg; joints [9.194, -75.733, 121.609, -46.593, 7.956, 53.486]
  MoveL 1032 to (-890, 800, 50) mm, rotated rx -180 ry 0 rz 90 deg; joints [9.194, -77.913, 120.983, -35.023, 10.091, 41.774]
  MoveL 1033 to (-890, 850, 50) mm, rotated rx -180 ry 0 rz 90 deg; joints [9.524, -80.005, 123.62, -37.744, 9.794, 44.766]
  MoveL 1034 to (-890, 850, -0.5) mm, rotated rx -180 ry 0 rz 90 deg; joints [9.524, -77.732, 124.267, -51.056, 7.694, 58.231]
  MoveL 1035 to (-890, 850, 50) mm, rotated rx -180 ry 0 rz 90 deg; joints [9.524, -80.005, 123.62, -37.744, 9.794, 44.766]
  MoveL 1036 to (-890, 900, 50) mm, rotated rx 180 ry 0 rz 90 deg; joints [9.877, -82.145, 126.217, -40.339, 9.6, 47.647]
  MoveL 1037 to (-890, 900, -0.5) mm, rotated rx 180 ry 0 rz 90 deg; joints [9.877, -79.772, 126.886, -55.347, 7.541, 62.82]
  MoveL 1038 to (-890, 900, 50) mm, rotated rx 180 ry 0 rz 90 deg; joints [9.877, -82.145, 126.217, -40.339, 9.6, 47.647]
  MoveL 1039 to (-890, 950, 50) mm, rotated rx 180 ry 0 rz 90 deg; joints [10.258, -84.343, 128.773, -42.695, 9.513, 50.306]
  MoveL 1040 to (-890, 950, -0.5) mm, rotated rx 180 ry 0 rz 90 deg; joints [10.258, -81.864, 129.467, -59.25, 7.493, 67.04]
  MoveL 1041 to (-890, 950, 50) mm, rotated rx 180 ry 0 rz 90 deg; joints [10.258, -84.343, 128.773, -42.695, 9.513, 50.306]
  MoveL 1042 to (-890, 1000, 50) mm, rotated rx 180 ry 0 rz 90 deg; joints [10.668, -86.612, 131.29, -44.693, 9.535, 52.624]
  MoveL 1043 to (-890, 1000, -0.5) mm, rotated rx 180 ry 0 rz 90 deg; joints [10.668, -84.017, 132.013, -62.561, 7.543, 70.686]
  MoveL 1044 to (-890, 1000, 50) mm, rotated rx 180 ry 0 rz 90 deg; joints [10.668, -86.612, 131.29, -44.693, 9.535, 52.624]
  MoveL 1045 to (-890, 1050, 50) mm, rotated rx 180 ry 0 rz 90 deg; joints [11.113, -88.964, 133.769, -46.223, 9.671, 54.493]
  MoveL 1046 to (-890, 1050, -0.5) mm, rotated rx -180 ry 0 rz 90 deg; joints [11.113, -86.246, 134.524, -65.104, 7.685, 73.586]
  MoveL 1047 to (-890, 1050, 50) mm, rotated rx 180 ry 0 rz 90 deg; joints [11.113, -88.964, 133.769, -46.223, 9.671, 54.493]
  MoveL 1048 to (-890, 1100, 50) mm, rotated rx -180 ry 0 rz 90 deg; joints [11.595, -91.415, 136.209, -47.195, 9.928, 55.824]
  MoveL 1049 to (-890, 1100, -0.5) mm, rotated rx 180 ry 0 rz 90 deg; joints [11.595, -88.564, 137, -66.748, 7.913, 75.609]
  MoveL 1050 to (-890, 1100, 50) mm, rotated rx -180 ry 0 rz 90 deg; joints [11.595, -91.415, 136.209, -47.195, 9.928, 55.824]
  MoveL 1051 to (-890, 1150, 50) mm, rotated rx -180 ry 0 rz 90 deg; joints [12.121, -93.984, 138.609, -47.547, 10.317, 56.557]
  MoveL 1052 to (-890, 1150, -0.5) mm, rotated rx 180 ry 0 rz 90 deg; joints [12.121, -90.991, 139.441, -67.405, 8.229, 76.669]
  MoveL 1053 to (-890, 1150, 50) mm, rotated rx -180 ry 0 rz 90 deg; joints [12.121, -93.984, 138.609, -47.547, 10.317, 56.557]
  MoveL 1054 to (-890, 1200, 50) mm, rotated rx 180 ry 0 rz 90 deg; joints [12.696, -96.694, 140.969, -47.251, 10.856, 56.665]
  MoveL 1055 to (-890, 1200, -0.5) mm, rotated rx 180 ry 0 rz 90 deg; joints [12.696, -93.548, 141.846, -67.028, 8.64, 76.722]
  MoveL 1056 to (-890, 1200, 50) mm, rotated rx 180 ry 0 rz 90 deg; joints [12.696, -96.694, 140.969, -47.251, 10.856, 56.665]
  MoveL 1057 to (-890, 1250, 50) mm, rotated rx 180 ry 0 rz 90 deg; joints [13.327, -99.571, 143.285, -46.32, 11.571, 56.163]
  MoveL 1058 to (-890, 1250, -0.5) mm, rotated rx -180 ry 0 rz 90 deg; joints [13.327, -96.263, 144.214, -65.612, 9.165, 75.765]
  MoveL 1059 to (-890, 1250, 50) mm, rotated rx 180 ry 0 rz 90 deg; joints [13.327, -99.571, 143.285, -46.32, 11.571, 56.163]
  MoveL 1060 to (-890, 1300, 50) mm, rotated rx 180 ry 0 rz 90 deg; joints [14.022, -102.648, 145.555, -44.803, 12.497, 55.1]
  MoveL 1061 to (-890, 1300, -0.5) mm, rotated rx 180 ry 0 rz 90 deg; joints [14.022, -99.169, 146.544, -63.199, 9.836, 73.84]
  MoveL 1062 to (-890, 1300, 50) mm, rotated rx 180 ry 0 rz 90 deg; joints [14.022, -102.648, 145.555, -44.803, 12.497, 55.1]
  MoveL 1063 to (-890, 1350, 50) mm, rotated rx -180 ry 0 rz 90 deg; joints [14.793, -105.964, 147.775, -42.787, 13.683, 53.564]
  MoveL 1064 to (-890, 1350, -0.5) mm, rotated rx -180 ry 0 rz 90 deg; joints [14.793, -102.307, 148.83, -59.886, 10.705, 71.045]
  MoveL 1065 to (-890, 1350, 50) mm, rotated rx -180 ry 0 rz 90 deg; joints [14.793, -105.964, 147.775, -42.787, 13.683, 53.564]
  MoveL 1066 to (-890, 1400, 50) mm, rotated rx -180 ry 0 rz 90 deg; joints [15.651, -109.567, 149.937, -40.388, 15.19, 51.668]
  MoveL 1067 to (-890, 1400, -0.5) mm, rotated rx -180 ry 0 rz 90 deg; joints [15.651, -105.731, 151.069, -55.83, 11.841, 67.539]
  MoveL 1068 to (-890, 1400, 50) mm, rotated rx -180 ry 0 rz 90 deg; joints [15.651, -109.567, 149.937, -40.388, 15.19, 51.668]
  MoveL 1069 to (-890, 1450, 50) mm, rotated rx -180 ry 0 rz 90 deg; joints [16.612, -113.514, 152.034, -37.739, 17.094, 49.547]
  MoveL 1070 to (-890, 1450, -0.5) mm, rotated rx -180 ry 0 rz 90 deg; joints [16.612, -109.505, 153.254, -51.254, 13.337, 63.54]
  MoveL 1071 to (-890, 1450, 50) mm, rotated rx -180 ry 0 rz 90 deg; joints [16.612, -113.514, 152.034, -37.739, 17.094, 49.547]
  MoveL 1072 to (-960, 50, 50) mm, rotated rx -180 ry 0 rz 90 deg; joints [7.868, -47.076, 73.298, -11.545, 25.494, 16.577]
  MoveL 1073 to (-960, 50, -0.5) mm, rotated rx 180 ry 0 rz 90 deg; joints [7.868, -45.813, 73.839, -12.361, 23.73, 17.474]
  MoveL 1074 to (-960, 50, 50) mm, rotated rx -180 ry 0 rz 90 deg; joints [7.868, -47.076, 73.298, -11.545, 25.494, 16.577]
  MoveL 1075 to (-960, 100, 50) mm, rotated rx 180 ry 0 rz 90 deg; joints [8.051, -49.289, 77.128, -12.541, 23.948, 17.764]
  MoveL 1076 to (-960, 100, -0.5) mm, rotated rx 180 ry 0 rz 90 deg; joints [8.051, -47.982, 77.66, -13.516, 22.155, 18.824]
  MoveL 1077 to (-960, 100, 50) mm, rotated rx 180 ry 0 rz 90 deg; joints [8.051, -49.289, 77.128, -12.541, 23.948, 17.764]
  MoveL 1078 to (-960, 150, 50) mm, rotated rx 180 ry 0 rz 90 deg; joints [8.243, -51.44, 80.804, -13.637, 22.5, 19.057]
  MoveL 1079 to (-960, 150, -0.5) mm, rotated rx 180 ry 0 rz 90 deg; joints [8.243, -50.087, 81.331, -14.804, 20.677, 20.312]
  MoveL 1080 to (-960, 150, 50) mm, rotated rx 180 ry 0 rz 90 deg; joints [8.243, -51.44, 80.804, -13.637, 22.5, 19.057]
  MoveL 1081 to (-960, 200, 50) mm, rotated rx 180 ry 0 rz 90 deg; joints [8.444, -53.539, 84.347, -14.844, 21.143, 20.466]
  MoveL 1082 to (-960, 200, -0.5) mm, rotated rx -180 ry 0 rz 90 deg; joints [8.444, -52.139, 84.871, -16.245, 19.289, 21.958]
  MoveL 1083 to (-960, 200, 50) mm, rotated rx 180 ry 0 rz 90 deg; joints [8.444, -53.539, 84.347, -14.844, 21.143, 20.466]
  MoveL 1084 to (-960, 250, 50) mm, rotated rx -180 ry 0 rz 90 deg; joints [8.655, -55.595, 87.772, -16.176, 19.872, 22.005]
  MoveL 1085 to (-960, 250, -0.5) mm, rotated rx -180 ry 0 rz 90 deg; joints [8.655, -54.148, 88.296, -17.858, 17.987, 23.784]
  MoveL 1086 to (-960, 250, 50) mm, rotated rx -180 ry 0 rz 90 deg; joints [8.655, -55.595, 87.772, -16.176, 19.872, 22.005]
  MoveL 1087 to (-960, 300, 50) mm, rotated rx -180 ry 0 rz 90 deg; joints [8.876, -57.618, 91.093, -17.646, 18.684, 23.689]
  MoveL 1088 to (-960, 300, -0.5) mm, rotated rx 180 ry 0 rz 90 deg; joints [8.876, -56.121, 91.618, -19.669, 16.768, 25.813]
  MoveL 1089 to (-960, 300, 50) mm, rotated rx -180 ry 0 rz 90 deg; joints [8.876, -57.618, 91.093, -17.646, 18.684, 23.689]
  MoveL 1090 to (-960, 350, 50) mm, rotated rx -180 ry 0 rz 90 deg; joints [9.11, -59.614, 94.321, -19.265, 17.577, 25.531]
  MoveL 1091 to (-960, 350, -0.5) mm, rotated rx -180 ry 0 rz 90 deg; joints [9.11, -58.066, 94.848, -21.701, 15.632, 28.073]
  MoveL 1092 to (-960, 350, 50) mm, rotated rx -180 ry 0 rz 90 deg; joints [9.11, -59.614, 94.321, -19.265, 17.577, 25.531]
  MoveL 1093 to (-960, 400, 50) mm, rotated rx 180 ry 0 rz 90 deg; joints [9.355, -61.59, 97.464, -21.047, 16.55, 27.543]
  MoveL 1094 to (-960, 400, -0.5) mm, rotated rx -180 ry 0 rz 90 deg; joints [9.355, -59.987, 97.995, -23.981, 14.579, 30.588]
  MoveL 1095 to (-960, 400, 50) mm, rotated rx 180 ry 0 rz 90 deg; joints [9.355, -61.59, 97.464, -21.047, 16.55, 27.543]
  MoveL 1096 to (-960, 450, 50) mm, rotated rx 180 ry 0 rz 90 deg; joints [9.615, -63.552, 100.53, -23.001, 15.605, 29.737]
  MoveL 1097 to (-960, 450, -0.5) mm, rotated rx -180 ry 0 rz 90 deg; joints [9.615, -61.893, 101.067, -26.532, 13.61, 33.385]
  MoveL 1098 to (-960, 450, 50) mm, rotated rx 180 ry 0 rz 90 deg; joints [9.615, -63.552, 100.53, -23.001, 15.605, 29.737]
  MoveL 1099 to (-960, 500, 50) mm, rotated rx -180 ry 0 rz 90 deg; joints [9.889, -65.506, 103.526, -25.133, 14.742, 32.119]
  MoveL 1100 to (-960, 500, -0.5) mm, rotated rx 180 ry 0 rz 90 deg; joints [9.889, -63.787, 104.07, -29.374, 12.729, 36.483]
  MoveL 1101 to (-960, 500, 50) mm, rotated rx -180 ry 0 rz 90 deg; joints [9.889, -65.506, 103.526, -25.133, 14.742, 32.119]
  MoveL 1102 to (-960, 550, 50) mm, rotated rx 180 ry 0 rz 90 deg; joints [10.178, -67.457, 106.457, -27.444, 13.963, 34.69]
  MoveL 1103 to (-960, 550, -0.5) mm, rotated rx 180 ry 0 rz 90 deg; joints [10.178, -65.675, 107.01, -32.518, 11.939, 39.896]
  MoveL 1104 to (-960, 550, 50) mm, rotated rx 180 ry 0 rz 90 deg; joints [10.178, -67.457, 106.457, -27.444, 13.963, 34.69]
  MoveL 1105 to (-960, 600, 50) mm, rotated rx -180 ry 0 rz 90 deg; joints [10.486, -69.411, 109.328, -29.925, 13.272, 37.444]
  MoveL 1106 to (-960, 600, -0.5) mm, rotated rx 180 ry 0 rz 90 deg; joints [10.486, -67.563, 109.891, -35.962, 11.246, 43.621]
  MoveL 1107 to (-960, 600, 50) mm, rotated rx -180 ry 0 rz 90 deg; joints [10.486, -69.411, 109.328, -29.925, 13.272, 37.444]
  MoveL 1108 to (-960, 650, 50) mm, rotated rx -180 ry 0 rz 90 deg; joints [10.812, -71.374, 112.144, -32.557, 12.672, 40.361]
  MoveL 1109 to (-960, 650, -0.5) mm, rotated rx 180 ry 0 rz 90 deg; joints [10.812, -69.456, 112.719, -39.682, 10.654, 47.635]
  MoveL 1110 to (-960, 650, 50) mm, rotated rx -180 ry 0 rz 90 deg; joints [10.812, -71.374, 112.144, -32.557, 12.672, 40.361]
  MoveL 1111 to (-960, 700, 50) mm, rotated rx 180 ry 0 rz 90 deg; joints [11.158, -73.351, 114.908, -35.305, 12.165, 43.409]
  MoveL 1112 to (-960, 700, -0.5) mm, rotated rx -180 ry 0 rz 90 deg; joints [11.158, -71.358, 115.496, -43.626, 10.167, 51.888]
  MoveL 1113 to (-960, 700, 50) mm, rotated rx 180 ry 0 rz 90 deg; joints [11.158, -73.351, 114.908, -35.305, 12.165, 43.409]
  MoveL 1114 to (-960, 750, 50) mm, rotated rx -180 ry 0 rz 90 deg; joints [11.527, -75.35, 117.622, -38.12, 11.755, 46.538]
  MoveL 1115 to (-960, 750, -0.5) mm, rotated rx 180 ry 0 rz 90 deg; joints [11.527, -73.277, 118.226, -47.711, 9.788, 56.299]
  MoveL 1116 to (-960, 750, 50) mm, rotated rx -180 ry 0 rz 90 deg; joints [11.527, -75.35, 117.622, -38.12, 11.755, 46.538]
  MoveL 1117 to (-960, 800, 50) mm, rotated rx 180 ry 0 rz 90 deg; joints [11.922, -77.376, 120.29, -40.935, 11.444, 49.684]
  MoveL 1118 to (-960, 800, -0.5) mm, rotated rx -180 ry 0 rz 90 deg; joints [11.922, -75.219, 120.911, -51.824, 9.519, 60.755]
  MoveL 1119 to (-960, 800, 50) mm, rotated rx 180 ry 0 rz 90 deg; joints [11.922, -77.376, 120.29, -40.935, 11.444, 49.684]
  MoveL 1120 to (-960, 850, 50) mm, rotated rx 180 ry 0 rz 90 deg; joints [12.343, -79.437, 122.914, -43.669, 11.235, 52.767]
  MoveL 1121 to (-960, 850, -0.5) mm, rotated rx 180 ry 0 rz 90 deg; joints [12.343, -77.19, 123.555, -55.826, 9.358, 65.12]
  MoveL 1122 to (-960, 850, 50) mm, rotated rx 180 ry 0 rz 90 deg; joints [12.343, -79.437, 122.914, -43.669, 11.235, 52.767]
  MoveL 1123 to (-960, 900, 50) mm, rotated rx 180 ry 0 rz 90 deg; joints [12.795, -81.542, 125.495, -46.23, 11.128, 55.696]
  MoveL 1124 to (-960, 900, -0.5) mm, rotated rx 180 ry 0 rz 90 deg; joints [12.795, -79.197, 126.158, -59.569, 9.302, 69.247]
  MoveL 1125 to (-960, 900, 50) mm, rotated rx 180 ry 0 rz 90 deg; joints [12.795, -81.542, 125.495, -46.23, 11.128, 55.696]
  MoveL 1126 to (-960, 950, 50) mm, rotated rx -180 ry 0 rz 90 deg; joints [13.281, -83.699, 128.035, -48.524, 11.126, 58.379]
  MoveL 1127 to (-960, 950, -0.5) mm, rotated rx 180 ry 0 rz 90 deg; joints [13.281, -81.251, 128.722, -62.907, 9.346, 72.991]
  MoveL 1128 to (-960, 950, 50) mm, rotated rx -180 ry 0 rz 90 deg; joints [13.281, -83.699, 128.035, -48.524, 11.126, 58.379]
  MoveL 1129 to (-960, 1000, 50) mm, rotated rx -180 ry 0 rz 90 deg; joints [13.805, -85.918, 130.534, -50.459, 11.229, 60.725]
  MoveL 1130 to (-960, 1000, -0.5) mm, rotated rx 180 ry 0 rz 90 deg; joints [13.805, -83.36, 131.248, -65.712, 9.483, 76.226]
  MoveL 1131 to (-960, 1000, 50) mm, rotated rx -180 ry 0 rz 90 deg; joints [13.805, -85.918, 130.534, -50.459, 11.229, 60.725]
  MoveL 1132 to (-960, 1050, 50) mm, rotated rx 180 ry 0 rz 90 deg; joints [14.37, -88.213, 132.993, -51.955, 11.439, 62.657]
  MoveL 1133 to (-960, 1050, -0.5) mm, rotated rx 180 ry 0 rz 90 deg; joints [14.37, -85.535, 133.737, -67.878, 9.707, 78.849]
  MoveL 1134 to (-960, 1050, 50) mm, rotated rx 180 ry 0 rz 90 deg; joints [14.37, -88.213, 132.993, -51.955, 11.439, 62.657]
  MoveL 1135 to (-960, 1100, 50) mm, rotated rx 180 ry 0 rz 90 deg; joints [14.983, -90.597, 135.411, -52.948, 11.763, 64.111]
  MoveL 1136 to (-960, 1100, -0.5) mm, rotated rx 180 ry 0 rz 90 deg; joints [14.983, -87.791, 136.19, -69.33, 10.014, 80.787]
  MoveL 1137 to (-960, 1100, 50) mm, rotated rx 180 ry 0 rz 90 deg; joints [14.983, -90.597, 135.411, -52.948, 11.763, 64.111]
  MoveL 1138 to (-960, 1150, 50) mm, rotated rx 180 ry 0 rz 90 deg; joints [15.649, -93.086, 137.789, -53.393, 12.208, 65.045]
  MoveL 1139 to (-960, 1150, -0.5) mm, rotated rx 180 ry 0 rz 90 deg; joints [15.649, -90.143, 138.606, -70.015, 10.407, 81.99]
  MoveL 1140 to (-960, 1150, 50) mm, rotated rx 180 ry 0 rz 90 deg; joints [15.649, -93.086, 137.789, -53.393, 12.208, 65.045]
  MoveL 1141 to (-960, 1200, 50) mm, rotated rx 180 ry 0 rz 90 deg; joints [16.375, -95.7, 140.124, -53.269, 12.79, 65.44]
  MoveL 1142 to (-960, 1200, -0.5) mm, rotated rx -180 ry 0 rz 90 deg; joints [16.375, -92.61, 140.984, -69.906, 10.89, 82.431]
  MoveL 1143 to (-960, 1200, 50) mm, rotated rx 180 ry 0 rz 90 deg; joints [16.375, -95.7, 140.124, -53.269, 12.79, 65.44]
  MoveL 1144 to (-960, 1250, 50) mm, rotated rx 180 ry 0 rz 90 deg; joints [17.17, -98.461, 142.414, -52.58, 13.528, 65.301]
  MoveL 1145 to (-960, 1250, -0.5) mm, rotated rx -180 ry 0 rz 90 deg; joints [17.17, -95.215, 143.323, -68.993, 11.479, 82.105]
  MoveL 1146 to (-960, 1250, 50) mm, rotated rx 180 ry 0 rz 90 deg; joints [17.17, -98.461, 142.414, -52.58, 13.528, 65.301]
  MoveL 1147 to (-960, 1300, 50) mm, rotated rx 180 ry 0 rz 90 deg; joints [18.043, -101.395, 144.656, -51.353, 14.453, 64.658]
  MoveL 1148 to (-960, 1300, -0.5) mm, rotated rx 180 ry 0 rz 90 deg; joints [18.043, -97.985, 145.62, -67.293, 12.199, 81.03]
  MoveL 1149 to (-960, 1300, 50) mm, rotated rx 180 ry 0 rz 90 deg; joints [18.043, -101.395, 144.656, -51.353, 14.453, 64.658]
  MoveL 1150 to (-960, 1350, 50) mm, rotated rx 180 ry 0 rz 90 deg; joints [19.007, -104.536, 146.847, -49.643, 15.602, 63.564]
  MoveL 1151 to (-960, 1350, -0.5) mm, rotated rx 180 ry 0 rz 90 deg; joints [19.007, -100.955, 147.873, -64.847, 13.087, 79.249]
  MoveL 1152 to (-960, 1350, 50) mm, rotated rx 180 ry 0 rz 90 deg; joints [19.007, -104.536, 146.847, -49.643, 15.602, 63.564]
  MoveL 1153 to (-960, 1400, 50) mm, rotated rx -180 ry 0 rz 90 deg; joints [20.074, -107.922, 148.98, -47.527, 17.029, 62.1]
  MoveL 1154 to (-960, 1400, -0.5) mm, rotated rx 180 ry 0 rz 90 deg; joints [20.074, -104.165, 150.077, -61.732, 14.197, 76.839]
  MoveL 1155 to (-960, 1400, 50) mm, rotated rx -180 ry 0 rz 90 deg; joints [20.074, -107.922, 148.98, -47.527, 17.029, 62.1]
  MoveL 1156 to (-960, 1450, 50) mm, rotated rx -180 ry 0 rz 90 deg; joints [21.263, -111.596, 151.049, -45.104, 18.794, 60.361]
  MoveL 1157 to (-960, 1450, -0.5) mm, rotated rx -180 ry 0 rz 90 deg; joints [21.263, -107.668, 152.226, -58.064, 15.6, 73.917]
  MoveL 1158 to (-960, 1450, 50) mm, rotated rx -180 ry 0 rz 90 deg; joints [21.263, -111.596, 151.049, -45.104, 18.794, 60.361]
  MoveL 1159 to (-1030, 50, 50) mm, rotated rx 180 ry 0 rz 90 deg; joints [9.672, -46.589, 72.451, -13.854, 26.203, 20.023]
  MoveL 1160 to (-1030, 50, -0.5) mm, rotated rx 180 ry 0 rz 90 deg; joints [9.672, -45.336, 72.993, -14.793, 24.463, 21.061]
  MoveL 1161 to (-1030, 50, 50) mm, rotated rx 180 ry 0 rz 90 deg; joints [9.672, -46.589, 72.451, -13.854, 26.203, 20.023]
  MoveL 1162 to (-1030, 100, 50) mm, rotated rx 180 ry 0 rz 90 deg; joints [9.896, -48.807, 76.297, -15.014, 24.676, 21.418]
  MoveL 1163 to (-1030, 100, -0.5) mm, rotated rx 180 ry 0 rz 90 deg; joints [9.896, -47.509, 76.831, -16.13, 22.911, 22.637]
  MoveL 1164 to (-1030, 100, 50) mm, rotated rx 180 ry 0 rz 90 deg; joints [9.896, -48.807, 76.297, -15.014, 24.676, 21.418]
  MoveL 1165 to (-1030, 150, 50) mm, rotated rx 180 ry 0 rz 90 deg; joints [10.13, -50.959, 79.986, -16.283, 23.251, 22.927]
  MoveL 1166 to (-1030, 150, -0.5) mm, rotated rx 180 ry 0 rz 90 deg; joints [10.13, -49.616, 80.514, -17.609, 21.461, 24.361]
  MoveL 1167 to (-1030, 150, 50) mm, rotated rx 180 ry 0 rz 90 deg; joints [10.13, -50.959, 79.986, -16.283, 23.251, 22.927]
  MoveL 1168 to (-1030, 200, 50) mm, rotated rx -180 ry 0 rz 90 deg; joints [10.375, -53.057, 83.538, -17.671, 21.923, 24.563]
  MoveL 1169 to (-1030, 200, -0.5) mm, rotated rx 180 ry 0 rz 90 deg; joints [10.375, -51.668, 84.063, -19.249, 20.107, 26.253]
  MoveL 1170 to (-1030, 200, 50) mm, rotated rx -180 ry 0 rz 90 deg; joints [10.375, -53.057, 83.538, -17.671, 21.923, 24.563]
  MoveL 1171 to (-1030, 250, 50) mm, rotated rx 180 ry 0 rz 90 deg; joints [10.632, -55.111, 86.97, -19.191, 20.685, 26.337]
  MoveL 1172 to (-1030, 250, -0.5) mm, rotated rx 180 ry 0 rz 90 deg; joints [10.632, -53.675, 87.493, -21.068, 18.845, 28.331]
  MoveL 1173 to (-1030, 250, 50) mm, rotated rx 180 ry 0 rz 90 deg; joints [10.632, -55.111, 86.97, -19.191, 20.685, 26.337]
  MoveL 1174 to (-1030, 300, 50) mm, rotated rx -180 ry 0 rz 90 deg; joints [10.902, -57.129, 90.294, -20.852, 19.535, 28.261]
  MoveL 1175 to (-1030, 300, -0.5) mm, rotated rx -180 ry 0 rz 90 deg; joints [10.902, -55.644, 90.818, -23.085, 17.672, 30.617]
  MoveL 1176 to (-1030, 300, 50) mm, rotated rx -180 ry 0 rz 90 deg; joints [10.902, -57.129, 90.294, -20.852, 19.535, 28.261]
  MoveL 1177 to (-1030, 350, 50) mm, rotated rx 180 ry 0 rz 90 deg; joints [11.187, -59.118, 93.523, -22.666, 18.471, 30.345]
  MoveL 1178 to (-1030, 350, -0.5) mm, rotated rx -180 ry 0 rz 90 deg; joints [11.187, -57.582, 94.049, -25.32, 16.587, 33.129]
  MoveL 1179 to (-1030, 350, 50) mm, rotated rx 180 ry 0 rz 90 deg; joints [11.187, -59.118, 93.523, -22.666, 18.471, 30.345]
  MoveL 1180 to (-1030, 400, 50) mm, rotated rx 180 ry 0 rz 90 deg; joints [11.486, -61.085, 96.665, -24.638, 17.493, 32.599]
  MoveL 1181 to (-1030, 400, -0.5) mm, rotated rx -180 ry 0 rz 90 deg; joints [11.486, -59.496, 97.195, -27.79, 15.592, 35.887]
  MoveL 1182 to (-1030, 400, 50) mm, rotated rx 180 ry 0 rz 90 deg; joints [11.486, -61.085, 96.665, -24.638, 17.493, 32.599]
  MoveL 1183 to (-1030, 450, 50) mm, rotated rx 180 ry 0 rz 90 deg; joints [11.801, -63.036, 99.728, -26.774, 16.601, 35.028]
  MoveL 1184 to (-1030, 450, -0.5) mm, rotated rx 180 ry 0 rz 90 deg; joints [11.801, -61.391, 100.263, -30.505, 14.687, 38.902]
  MoveL 1185 to (-1030, 450, 50) mm, rotated rx 180 ry 0 rz 90 deg; joints [11.801, -63.036, 99.728, -26.774, 16.601, 35.028]
  MoveL 1186 to (-1030, 500, 50) mm, rotated rx 180 ry 0 rz 90 deg; joints [12.134, -64.976, 102.719, -29.073, 15.797, 37.632]
  MoveL 1187 to (-1030, 500, -0.5) mm, rotated rx -180 ry 0 rz 90 deg; joints [12.134, -63.274, 103.261, -33.473, 13.877, 42.182]
  MoveL 1188 to (-1030, 500, 50) mm, rotated rx 180 ry 0 rz 90 deg; joints [12.134, -64.976, 102.719, -29.073, 15.797, 37.632]
  MoveL 1189 to (-1030, 550, 50) mm, rotated rx 180 ry 0 rz 90 deg; joints [12.486, -66.911, 105.644, -31.527, 15.082, 40.403]
  MoveL 1190 to (-1030, 550, -0.5) mm, rotated rx 180 ry 0 rz 90 deg; joints [12.486, -65.148, 106.194, -36.686, 13.164, 45.722]
  MoveL 1191 to (-1030, 550, 50) mm, rotated rx 180 ry 0 rz 90 deg; joints [12.486, -66.911, 105.644, -31.527, 15.082, 40.403]
  MoveL 1192 to (-1030, 600, 50) mm, rotated rx 180 ry 0 rz 90 deg; joints [12.858, -68.847, 108.507, -34.118, 14.459, 43.326]
  MoveL 1193 to (-1030, 600, -0.5) mm, rotated rx 180 ry 0 rz 90 deg; joints [12.858, -67.019, 109.067, -40.123, 12.552, 49.5]
  MoveL 1194 to (-1030, 600, 50) mm, rotated rx 180 ry 0 rz 90 deg; joints [12.858, -68.847, 108.507, -34.118, 14.459, 43.326]
  MoveL 1195 to (-1030, 650, 50) mm, rotated rx 180 ry 0 rz 90 deg; joints [13.253, -70.789, 111.313, -36.819, 13.93, 46.375]
  MoveL 1196 to (-1030, 650, -0.5) mm, rotated rx 180 ry 0 rz 90 deg; joints [13.253, -68.892, 111.884, -43.743, 12.044, 53.479]
  MoveL 1197 to (-1030, 650, 50) mm, rotated rx 180 ry 0 rz 90 deg; joints [13.253, -70.789, 111.313, -36.819, 13.93, 46.375]
  MoveL 1198 to (-1030, 700, 50) mm, rotated rx 180 ry 0 rz 90 deg; joints [13.673, -72.743, 114.065, -39.59, 13.499, 49.51]
  MoveL 1199 to (-1030, 700, -0.5) mm, rotated rx 180 ry 0 rz 90 deg; joints [13.673, -70.773, 114.649, -47.485, 11.643, 57.597]
  MoveL 1200 to (-1030, 700, 50) mm, rotated rx 180 ry 0 rz 90 deg; joints [13.673, -72.743, 114.065, -39.59, 13.499, 49.51]
  MoveL 1201 to (-1030, 750, 50) mm, rotated rx -180 ry 0 rz 90 deg; joints [14.119, -74.713, 116.766, -42.378, 13.165, 52.68]
  MoveL 1202 to (-1030, 750, -0.5) mm, rotated rx 180 ry 0 rz 90 deg; joints [14.119, -72.667, 117.365, -51.267, 11.35, 61.775]
  MoveL 1203 to (-1030, 750, 50) mm, rotated rx -180 ry 0 rz 90 deg; joints [14.119, -74.713, 116.766, -42.378, 13.165, 52.68]
  MoveL 1204 to (-1030, 800, 50) mm, rotated rx 180 ry 0 rz 90 deg; joints [14.595, -76.707, 119.42, -45.12, 12.932, 55.824]
  MoveL 1205 to (-1030, 800, -0.5) mm, rotated rx -180 ry 0 rz 90 deg; joints [14.595, -74.579, 120.035, -54.989, 11.164, 65.913]
  MoveL 1206 to (-1030, 800, 50) mm, rotated rx 180 ry 0 rz 90 deg; joints [14.595, -76.707, 119.42, -45.12, 12.932, 55.824]
  MoveL 1207 to (-1030, 850, 50) mm, rotated rx -180 ry 0 rz 90 deg; joints [15.104, -78.732, 122.027, -47.744, 12.8, 58.871]
  MoveL 1208 to (-1030, 850, -0.5) mm, rotated rx 180 ry 0 rz 90 deg; joints [15.104, -76.516, 122.661, -58.544, 11.083, 69.907]
  MoveL 1209 to (-1030, 850, 50) mm, rotated rx -180 ry 0 rz 90 deg; joints [15.104, -78.732, 122.027, -47.744, 12.8, 58.871]
  MoveL 1210 to (-1030, 900, 50) mm, rotated rx -180 ry 0 rz 90 deg; joints [15.648, -80.794, 124.59, -50.176, 12.769, 61.749]
  MoveL 1211 to (-1030, 900, -0.5) mm, rotated rx -180 ry 0 rz 90 deg; joints [15.648, -78.485, 125.244, -61.821, 11.102, 73.649]
  MoveL 1212 to (-1030, 900, 50) mm, rotated rx -180 ry 0 rz 90 deg; joints [15.648, -80.794, 124.59, -50.176, 12.769, 61.749]
  MoveL 1213 to (-1030, 950, 50) mm, rotated rx 180 ry 0 rz 90 deg; joints [16.231, -82.902, 127.109, -52.34, 12.838, 64.384]
  MoveL 1214 to (-1030, 950, -0.5) mm, rotated rx -180 ry 0 rz 90 deg; joints [16.231, -80.493, 127.787, -64.722, 11.218, 77.041]
  MoveL 1215 to (-1030, 950, 50) mm, rotated rx 180 ry 0 rz 90 deg; joints [16.231, -82.902, 127.109, -52.34, 12.838, 64.384]
  MoveL 1216 to (-1030, 1000, 50) mm, rotated rx -180 ry 0 rz 90 deg; joints [16.859, -85.064, 129.586, -54.169, 13.01, 66.711]
  MoveL 1217 to (-1030, 1000, -0.5) mm, rotated rx 180 ry 0 rz 90 deg; joints [16.859, -82.549, 130.29, -67.161, 11.423, 80]
  MoveL 1218 to (-1030, 1000, 50) mm, rotated rx -180 ry 0 rz 90 deg; joints [16.859, -85.064, 129.586, -54.169, 13.01, 66.711]
  MoveL 1219 to (-1030, 1050, 50) mm, rotated rx -180 ry 0 rz 90 deg; joints [17.536, -87.292, 132.021, -55.604, 13.285, 68.673]
  MoveL 1220 to (-1030, 1050, -0.5) mm, rotated rx 180 ry 0 rz 90 deg; joints [17.536, -84.662, 132.753, -69.071, 11.713, 82.462]
  MoveL 1221 to (-1030, 1050, 50) mm, rotated rx -180 ry 0 rz 90 deg; joints [17.536, -87.292, 132.021, -55.604, 13.285, 68.673]
  MoveL 1222 to (-1030, 1100, 50) mm, rotated rx -180 ry 0 rz 90 deg; joints [18.267, -89.597, 134.414, -56.6, 13.667, 70.227]
  MoveL 1223 to (-1030, 1100, -0.5) mm, rotated rx -180 ry 0 rz 90 deg; joints [18.267, -86.845, 135.178, -70.402, 12.086, 84.38]
  MoveL 1224 to (-1030, 1100, 50) mm, rotated rx -180 ry 0 rz 90 deg; joints [18.267, -89.597, 134.414, -56.6, 13.667, 70.227]
  MoveL 1225 to (-1030, 1150, 50) mm, rotated rx 180 ry 0 rz 90 deg; joints [19.06, -91.993, 136.763, -57.125, 14.163, 71.343]
  MoveL 1226 to (-1030, 1150, -0.5) mm, rotated rx 180 ry 0 rz 90 deg; joints [19.06, -89.111, 137.563, -71.123, 12.544, 85.724]
  MoveL 1227 to (-1030, 1150, 50) mm, rotated rx 180 ry 0 rz 90 deg; joints [19.06, -91.993, 136.763, -57.125, 14.163, 71.343]
  MoveL 1228 to (-1030, 1200, 50) mm, rotated rx -180 ry 0 rz 90 deg; joints [19.921, -94.496, 139.068, -57.165, 14.785, 72.009]
  MoveL 1229 to (-1030, 1200, -0.5) mm, rotated rx -180 ry 0 rz 90 deg; joints [19.921, -91.474, 139.908, -71.214, 13.091, 86.478]
  MoveL 1230 to (-1030, 1200, 50) mm, rotated rx -180 ry 0 rz 90 deg; joints [19.921, -94.496, 139.068, -57.165, 14.785, 72.009]
  MoveL 1231 to (-1030, 1250, 50) mm, rotated rx -180 ry 0 rz 90 deg; joints [20.861, -97.123, 141.327, -56.718, 15.549, 72.227]
  MoveL 1232 to (-1030, 1250, -0.5) mm, rotated rx 180 ry 0 rz 90 deg; joints [20.861, -93.953, 142.212, -70.669, 13.738, 86.64]
  MoveL 1233 to (-1030, 1250, 50) mm, rotated rx -180 ry 0 rz 90 deg; joints [20.861, -97.123, 141.327, -56.718, 15.549, 72.227]
  MoveL 1234 to (-1030, 1300, 50) mm, rotated rx 180 ry 0 rz 90 deg; joints [21.888, -99.897, 143.536, -55.801, 16.479, 72.016]
  MoveL 1235 to (-1030, 1300, -0.5) mm, rotated rx -180 ry 0 rz 90 deg; joints [21.888, -96.571, 144.471, -69.496, 14.506, 86.22]
  MoveL 1236 to (-1030, 1300, 50) mm, rotated rx 180 ry 0 rz 90 deg; joints [21.888, -99.897, 143.536, -55.801, 16.479, 72.016]
  MoveL 1237 to (-1030, 1350, 50) mm, rotated rx -180 ry 0 rz 90 deg; joints [23.017, -102.842, 145.692, -54.45, 17.604, 71.411]
  MoveL 1238 to (-1030, 1350, -0.5) mm, rotated rx -180 ry 0 rz 90 deg; joints [23.017, -99.353, 146.684, -67.719, 15.422, 85.243]
  MoveL 1239 to (-1030, 1350, 50) mm, rotated rx -180 ry 0 rz 90 deg; joints [23.017, -102.842, 145.692, -54.45, 17.604, 71.411]
  MoveL 1240 to (-1030, 1400, 50) mm, rotated rx 180 ry 0 rz 90 deg; joints [24.261, -105.987, 147.79, -52.714, 18.966, 70.465]
  MoveL 1241 to (-1030, 1400, -0.5) mm, rotated rx -180 ry 0 rz 90 deg; joints [24.261, -102.33, 148.846, -65.378, 16.526, 83.753]
  MoveL 1242 to (-1030, 1400, 50) mm, rotated rx 180 ry 0 rz 90 deg; joints [24.261, -105.987, 147.79, -52.714, 18.966, 70.465]
  MoveL 1243 to (-1100, 50, 50) mm, rotated rx 180 ry 0 rz 90 deg; joints [11.457, -45.999, 71.42, -15.959, 27.043, 23.24]
  MoveL 1244 to (-1100, 50, -0.5) mm, rotated rx 180 ry 0 rz 90 deg; joints [11.457, -44.757, 71.966, -16.99, 25.329, 24.389]
  MoveL 1245 to (-1100, 50, 50) mm, rotated rx 180 ry 0 rz 90 deg; joints [11.457, -45.999, 71.42, -15.959, 27.043, 23.24]
  MoveL 1246 to (-1100, 100, 50) mm, rotated rx -180 ry 0 rz 90 deg; joints [11.72, -48.223, 75.288, -17.251, 25.534, 24.811]
  MoveL 1247 to (-1100, 100, -0.5) mm, rotated rx 180 ry 0 rz 90 deg; joints [11.72, -46.937, 75.824, -18.468, 23.8, 26.15]
  MoveL 1248 to (-1100, 100, 50) mm, rotated rx -180 ry 0 rz 90 deg; joints [11.72, -48.223, 75.288, -17.251, 25.534, 24.811]
  MoveL 1249 to (-1100, 150, 50) mm, rotated rx -180 ry 0 rz 90 deg; joints [11.995, -50.377, 78.994, -18.655, 24.134, 26.5]
  MoveL 1250 to (-1100, 150, -0.5) mm, rotated rx -180 ry 0 rz 90 deg; joints [11.995, -49.047, 79.523, -20.091, 22.379, 28.063]
  MoveL 1251 to (-1100, 150, 50) mm, rotated rx -180 ry 0 rz 90 deg; joints [11.995, -50.377, 78.994, -18.655, 24.134, 26.5]
  MoveL 1252 to (-1100, 200, 50) mm, rotated rx 180 ry 0 rz 90 deg; joints [12.283, -52.475, 82.558, -20.181, 22.834, 28.317]
  MoveL 1253 to (-1100, 200, -0.5) mm, rotated rx -180 ry 0 rz 90 deg; joints [12.283, -51.1, 83.083, -21.874, 21.059, 30.143]
  MoveL 1254 to (-1100, 200, 50) mm, rotated rx 180 ry 0 rz 90 deg; joints [12.283, -52.475, 82.558, -20.181, 22.834, 28.317]
  MoveL 1255 to (-1100, 250, 50) mm, rotated rx 180 ry 0 rz 90 deg; joints [12.585, -54.526, 85.997, -21.837, 21.631, 30.273]
  MoveL 1256 to (-1100, 250, -0.5) mm, rotated rx 180 ry 0 rz 90 deg; joints [12.585, -53.104, 86.521, -23.832, 19.837, 32.406]
  MoveL 1257 to (-1100, 250, 50) mm, rotated rx 180 ry 0 rz 90 deg; joints [12.585, -54.526, 85.997, -21.837, 21.631, 30.273]
  MoveL 1258 to (-1100, 300, 50) mm, rotated rx 180 ry 0 rz 90 deg; joints [12.901, -56.539, 89.327, -23.632, 20.519, 32.377]
  MoveL 1259 to (-1100, 300, -0.5) mm, rotated rx -180 ry 0 rz 90 deg; joints [12.901, -55.068, 89.851, -25.98, 18.709, 34.869]
  MoveL 1260 to (-1100, 300, 50) mm, rotated rx 180 ry 0 rz 90 deg; joints [12.901, -56.539, 89.327, -23.632, 20.519, 32.377]
  MoveL 1261 to (-1100, 350, 50) mm, rotated rx -180 ry 0 rz 90 deg; joints [13.234, -58.52, 92.558, -25.571, 19.499, 34.635]
  MoveL 1262 to (-1100, 350, -0.5) mm, rotated rx 180 ry 0 rz 90 deg; joints [13.234, -57, 93.083, -28.328, 17.675, 37.543]
  MoveL 1263 to (-1100, 350, 50) mm, rotated rx -180 ry 0 rz 90 deg; joints [13.234, -58.52, 92.558, -25.571, 19.499, 34.635]
  MoveL 1264 to (-1100, 400, 50) mm, rotated rx -180 ry 0 rz 90 deg; joints [13.584, -60.477, 95.699, -27.657, 18.569, 37.052]
  MoveL 1265 to (-1100, 400, -0.5) mm, rotated rx 180 ry 0 rz 90 deg; joints [13.584, -58.905, 96.228, -30.885, 16.735, 40.439]
  MoveL 1266 to (-1100, 400, 50) mm, rotated rx -180 ry 0 rz 90 deg; joints [13.584, -60.477, 95.699, -27.657, 18.569, 37.052]
  MoveL 1267 to (-1100, 450, 50) mm, rotated rx -180 ry 0 rz 90 deg; joints [13.953, -62.415, 98.76, -29.889, 17.729, 39.628]
  MoveL 1268 to (-1100, 450, -0.5) mm, rotated rx -180 ry 0 rz 90 deg; joints [13.953, -60.789, 99.293, -33.654, 15.892, 43.56]
  MoveL 1269 to (-1100, 450, 50) mm, rotated rx -180 ry 0 rz 90 deg; joints [13.953, -62.415, 98.76, -29.889, 17.729, 39.628]
  MoveL 1270 to (-1100, 500, 50) mm, rotated rx 180 ry 0 rz 90 deg; joints [14.342, -64.341, 101.746, -32.26, 16.981, 42.357]
  MoveL 1271 to (-1100, 500, -0.5) mm, rotated rx 180 ry 0 rz 90 deg; joints [14.342, -62.658, 102.285, -36.628, 15.146, 46.901]
  MoveL 1272 to (-1100, 500, 50) mm, rotated rx 180 ry 0 rz 90 deg; joints [14.342, -64.341, 101.746, -32.26, 16.981, 42.357]
  MoveL 1273 to (-1100, 550, 50) mm, rotated rx 180 ry 0 rz 90 deg; joints [14.752, -66.258, 104.663, -34.757, 16.326, 45.226]
  MoveL 1274 to (-1100, 550, -0.5) mm, rotated rx -180 ry 0 rz 90 deg; joints [14.752, -64.516, 105.211, -39.789, 14.502, 50.445]
  MoveL 1275 to (-1100, 550, 50) mm, rotated rx 180 ry 0 rz 90 deg; joints [14.752, -66.258, 104.663, -34.757, 16.326, 45.226]
  MoveL 1276 to (-1100, 600, 50) mm, rotated rx 180 ry 0 rz 90 deg; joints [15.187, -68.173, 107.517, -37.357, 15.766, 48.215]
  MoveL 1277 to (-1100, 600, -0.5) mm, rotated rx 180 ry 0 rz 90 deg; joints [15.187, -66.368, 108.074, -43.108, 13.96, 54.164]
  MoveL 1278 to (-1100, 600, 50) mm, rotated rx 180 ry 0 rz 90 deg; joints [15.187, -68.173, 107.517, -37.357, 15.766, 48.215]
  MoveL 1279 to (-1100, 650, 50) mm, rotated rx -180 ry 0 rz 90 deg; joints [15.647, -70.091, 110.312, -40.027, 15.302, 51.292]
  MoveL 1280 to (-1100, 650, -0.5) mm, rotated rx 180 ry 0 rz 90 deg; joints [15.647, -68.219, 110.879, -46.538, 13.524, 58.013]
  MoveL 1281 to (-1100, 650, 50) mm, rotated rx -180 ry 0 rz 90 deg; joints [15.647, -70.091, 110.312, -40.027, 15.302, 51.292]
  MoveL 1282 to (-1100, 700, 50) mm, rotated rx -180 ry 0 rz 90 deg; joints [16.135, -72.017, 113.051, -42.729, 14.936, 54.419]
  MoveL 1283 to (-1100, 700, -0.5) mm, rotated rx -180 ry 0 rz 90 deg; joints [16.135, -70.075, 113.63, -50.019, 13.193, 61.933]
  MoveL 1284 to (-1100, 700, 50) mm, rotated rx -180 ry 0 rz 90 deg; joints [16.135, -72.017, 113.051, -42.729, 14.936, 54.419]
  MoveL 1285 to (-1100, 750, 50) mm, rotated rx -180 ry 0 rz 90 deg; joints [16.653, -73.956, 115.738, -45.41, 14.67, 57.548]
  MoveL 1286 to (-1100, 750, -0.5) mm, rotated rx -180 ry 0 rz 90 deg; joints [16.653, -71.94, 116.331, -53.478, 12.969, 65.854]
  MoveL 1287 to (-1100, 750, 50) mm, rotated rx -180 ry 0 rz 90 deg; joints [16.653, -73.956, 115.738, -45.41, 14.67, 57.548]
  MoveL 1288 to (-1100, 800, 50) mm, rotated rx -180 ry 0 rz 90 deg; joints [17.205, -75.914, 118.374, -48.017, 14.503, 60.624]
  MoveL 1289 to (-1100, 800, -0.5) mm, rotated rx -180 ry 0 rz 90 deg; joints [17.205, -73.819, 118.982, -56.834, 12.849, 69.696]
  MoveL 1290 to (-1100, 800, 50) mm, rotated rx -180 ry 0 rz 90 deg; joints [17.205, -75.914, 118.374, -48.017, 14.503, 60.624]
  MoveL 1291 to (-1100, 850, 50) mm, rotated rx 180 ry 0 rz 90 deg; joints [17.794, -77.897, 120.962, -50.488, 14.435, 63.589]
  MoveL 1292 to (-1100, 850, -0.5) mm, rotated rx 180 ry 0 rz 90 deg; joints [17.794, -75.717, 121.588, -60.005, 12.83, 73.379]
  MoveL 1293 to (-1100, 850, 50) mm, rotated rx 180 ry 0 rz 90 deg; joints [17.794, -77.897, 120.962, -50.488, 14.435, 63.589]
  MoveL 1294 to (-1100, 900, 50) mm, rotated rx 180 ry 0 rz 90 deg; joints [18.423, -79.911, 123.504, -52.764, 14.466, 66.385]
  MoveL 1295 to (-1100, 900, -0.5) mm, rotated rx -180 ry 0 rz 90 deg; joints [18.423, -77.642, 124.149, -62.909, 12.908, 76.823]
  MoveL 1296 to (-1100, 900, 50) mm, rotated rx 180 ry 0 rz 90 deg; joints [18.423, -79.911, 123.504, -52.764, 14.466, 66.385]
  MoveL 1297 to (-1100, 950, 50) mm, rotated rx 180 ry 0 rz 90 deg; joints [19.096, -81.963, 126, -54.788, 14.595, 68.956]
  MoveL 1298 to (-1100, 950, -0.5) mm, rotated rx 180 ry 0 rz 90 deg; joints [19.096, -79.599, 126.667, -65.477, 13.079, 79.962]
  MoveL 1299 to (-1100, 950, 50) mm, rotated rx 180 ry 0 rz 90 deg; joints [19.096, -81.963, 126, -54.788, 14.595, 68.956]
  MoveL 1300 to (-1100, 1000, 50) mm, rotated rx -180 ry 0 rz 90 deg; joints [19.818, -84.062, 128.452, -56.507, 14.823, 71.255]
  MoveL 1301 to (-1100, 1000, -0.5) mm, rotated rx -180 ry 0 rz 90 deg; joints [19.818, -81.596, 129.143, -67.648, 13.338, 82.737]
  MoveL 1302 to (-1100, 1000, 50) mm, rotated rx -180 ry 0 rz 90 deg; joints [19.818, -84.062, 128.452, -56.507, 14.823, 71.255]
  MoveL 1303 to (-1100, 1050, 50) mm, rotated rx -180 ry 0 rz 90 deg; joints [20.595, -86.215, 130.859, -57.88, 15.151, 73.24]
  MoveL 1304 to (-1100, 1050, -0.5) mm, rotated rx 180 ry 0 rz 90 deg; joints [20.595, -83.641, 131.577, -69.376, 13.681, 85.106]
  MoveL 1305 to (-1100, 1050, 50) mm, rotated rx -180 ry 0 rz 90 deg; joints [20.595, -86.215, 130.859, -57.88, 15.151, 73.24]
  MoveL 1306 to (-1100, 1100, 50) mm, rotated rx -180 ry 0 rz 90 deg; joints [21.431, -88.434, 133.222, -58.874, 15.582, 74.881]
  MoveL 1307 to (-1100, 1100, -0.5) mm, rotated rx 180 ry 0 rz 90 deg; joints [21.431, -85.744, 133.97, -70.628, 14.108, 87.037]
  MoveL 1308 to (-1100, 1100, 50) mm, rotated rx -180 ry 0 rz 90 deg; joints [21.431, -88.434, 133.222, -58.874, 15.582, 74.881]
  MoveL 1309 to (-1100, 1150, 50) mm, rotated rx 180 ry 0 rz 90 deg; joints [22.335, -90.728, 135.54, -59.466, 16.121, 76.158]
  MoveL 1310 to (-1100, 1150, -0.5) mm, rotated rx 180 ry 0 rz 90 deg; joints [22.335, -87.915, 136.32, -71.381, 14.618, 88.511]
  MoveL 1311 to (-1100, 1150, 50) mm, rotated rx 180 ry 0 rz 90 deg; joints [22.335, -90.728, 135.54, -59.466, 16.121, 76.158]
  MoveL 1312 to (-1100, 1200, 50) mm, rotated rx 180 ry 0 rz 90 deg; joints [23.315, -93.11, 137.811, -59.644, 16.777, 77.063]
  MoveL 1313 to (-1100, 1200, -0.5) mm, rotated rx 180 ry 0 rz 90 deg; joints [23.315, -90.166, 138.628, -71.624, 15.216, 89.521]
  MoveL 1314 to (-1100, 1200, 50) mm, rotated rx 180 ry 0 rz 90 deg; joints [23.315, -93.11, 137.811, -59.644, 16.777, 77.063]
  MoveL 1315 to (-1100, 1250, 50) mm, rotated rx 180 ry 0 rz 90 deg; joints [24.379, -95.595, 140.033, -59.41, 17.563, 77.599]
  MoveL 1316 to (-1100, 1250, -0.5) mm, rotated rx 180 ry 0 rz 90 deg; joints [24.379, -92.511, 140.891, -71.353, 15.911, 90.065]
  MoveL 1317 to (-1100, 1250, 50) mm, rotated rx 180 ry 0 rz 90 deg; joints [24.379, -95.595, 140.033, -59.41, 17.563, 77.599]
  MoveL 1318 to (-1100, 1300, 50) mm, rotated rx -180 ry 0 rz 90 deg; joints [25.537, -98.198, 142.204, -58.772, 18.498, 77.778]
  MoveL 1319 to (-1100, 1300, -0.5) mm, rotated rx 180 ry 0 rz 90 deg; joints [25.537, -94.968, 143.108, -70.574, 16.719, 90.154]
  MoveL 1320 to (-1100, 1300, 50) mm, rotated rx -180 ry 0 rz 90 deg; joints [25.537, -98.198, 142.204, -58.772, 18.498, 77.778]
  MoveL 1321 to (-1100, 1350, 50) mm, rotated rx 180 ry 0 rz 90 deg; joints [26.803, -100.938, 144.32, -57.755, 19.604, 77.627]
  MoveL 1322 to (-1100, 1350, -0.5) mm, rotated rx 180 ry 0 rz 90 deg; joints [26.803, -97.554, 145.275, -69.302, 17.659, 89.806]
  MoveL 1323 to (-1100, 1350, 50) mm, rotated rx 180 ry 0 rz 90 deg; joints [26.803, -100.938, 144.32, -57.755, 19.604, 77.627]
  MoveL 1324 to (-1170, 50, 50) mm, rotated rx 180 ry 0 rz 90 deg; joints [13.22, -45.305, 70.203, -17.848, 28.007, 26.216]
  MoveL 1325 to (-1170, 50, -0.5) mm, rotated rx -180 ry 0 rz 90 deg; joints [13.22, -44.076, 70.752, -18.941, 26.32, 27.444]
  MoveL 1326 to (-1170, 50, 50) mm, rotated rx 180 ry 0 rz 90 deg; joints [13.22, -45.305, 70.203, -17.848, 28.007, 26.216]
  MoveL 1327 to (-1170, 100, 50) mm, rotated rx -180 ry 0 rz 90 deg; joints [13.521, -47.536, 74.099, -19.242, 26.516, 27.931]
  MoveL 1328 to (-1170, 100, -0.5) mm, rotated rx 180 ry 0 rz 90 deg; joints [13.521, -46.264, 74.637, -20.524, 24.813, 29.353]
  MoveL 1329 to (-1170, 100, 50) mm, rotated rx -180 ry 0 rz 90 deg; joints [13.521, -47.536, 74.099, -19.242, 26.516, 27.931]
  MoveL 1330 to (-1170, 150, 50) mm, rotated rx 180 ry 0 rz 90 deg; joints [13.835, -49.695, 77.825, -20.747, 25.138, 29.763]
  MoveL 1331 to (-1170, 150, -0.5) mm, rotated rx 180 ry 0 rz 90 deg; joints [13.835, -48.379, 78.356, -22.248, 23.419, 31.41]
  MoveL 1332 to (-1170, 150, 50) mm, rotated rx 180 ry 0 rz 90 deg; joints [13.835, -49.695, 77.825, -20.747, 25.138, 29.763]
  MoveL 1333 to (-1170, 200, 50) mm, rotated rx 180 ry 0 rz 90 deg; joints [14.163, -51.793, 81.404, -22.37, 23.866, 31.721]
  MoveL 1334 to (-1170, 200, -0.5) mm, rotated rx 180 ry 0 rz 90 deg; joints [14.163, -50.433, 81.931, -24.125, 22.132, 33.627]
  MoveL 1335 to (-1170, 200, 50) mm, rotated rx 180 ry 0 rz 90 deg; joints [14.163, -51.793, 81.404, -22.37, 23.866, 31.721]
  MoveL 1336 to (-1170, 250, 50) mm, rotated rx 180 ry 0 rz 90 deg; joints [14.508, -53.842, 84.855, -24.117, 22.695, 33.812]
  MoveL 1337 to (-1170, 250, -0.5) mm, rotated rx -180 ry 0 rz 90 deg; joints [14.508, -52.435, 85.379, -26.166, 20.947, 36.019]
  MoveL 1338 to (-1170, 250, 50) mm, rotated rx 180 ry 0 rz 90 deg; joints [14.508, -53.842, 84.855, -24.117, 22.695, 33.812]
  MoveL 1339 to (-1170, 300, 50) mm, rotated rx 180 ry 0 rz 90 deg; joints [14.869, -55.849, 88.191, -25.994, 21.621, 36.043]
  MoveL 1340 to (-1170, 300, -0.5) mm, rotated rx 180 ry 0 rz 90 deg; joints [14.869, -54.395, 88.715, -28.38, 19.862, 38.593]
  MoveL 1341 to (-1170, 300, 50) mm, rotated rx 180 ry 0 rz 90 deg; joints [14.869, -55.849, 88.191, -25.994, 21.621, 36.043]
  MoveL 1342 to (-1170, 350, 50) mm, rotated rx 180 ry 0 rz 90 deg; joints [15.248, -57.822, 91.426, -28.002, 20.641, 38.417]
  MoveL 1343 to (-1170, 350, -0.5) mm, rotated rx -180 ry 0 rz 90 deg; joints [15.248, -56.32, 91.95, -30.772, 18.875, 41.359]
  MoveL 1344 to (-1170, 350, 50) mm, rotated rx 180 ry 0 rz 90 deg; joints [15.248, -57.822, 91.426, -28.002, 20.641, 38.417]
  MoveL 1345 to (-1170, 400, 50) mm, rotated rx -180 ry 0 rz 90 deg; joints [15.646, -59.768, 94.568, -30.141, 19.756, 40.934]
  MoveL 1346 to (-1170, 400, -0.5) mm, rotated rx 180 ry 0 rz 90 deg; joints [15.646, -58.215, 95.095, -33.343, 17.986, 44.318]
  MoveL 1347 to (-1170, 400, 50) mm, rotated rx -180 ry 0 rz 90 deg; joints [15.646, -59.768, 94.568, -30.141, 19.756, 40.934]
  MoveL 1348 to (-1170, 450, 50) mm, rotated rx 180 ry 0 rz 90 deg; joints [16.065, -61.693, 97.626, -32.405, 18.964, 43.591]
  MoveL 1349 to (-1170, 450, -0.5) mm, rotated rx 180 ry 0 rz 90 deg; joints [16.065, -60.087, 98.157, -36.089, 17.197, 47.466]
  MoveL 1350 to (-1170, 450, 50) mm, rotated rx 180 ry 0 rz 90 deg; joints [16.065, -61.693, 97.626, -32.405, 18.964, 43.591]
  MoveL 1351 to (-1170, 500, 50) mm, rotated rx -180 ry 0 rz 90 deg; joints [16.507, -63.602, 100.607, -34.782, 18.268, 46.376]
  MoveL 1352 to (-1170, 500, -0.5) mm, rotated rx 180 ry 0 rz 90 deg; joints [16.507, -61.941, 101.144, -38.996, 16.509, 50.792]
  MoveL 1353 to (-1170, 500, 50) mm, rotated rx -180 ry 0 rz 90 deg; joints [16.507, -63.602, 100.607, -34.782, 18.268, 46.376]
  MoveL 1354 to (-1170, 550, 50) mm, rotated rx -180 ry 0 rz 90 deg; joints [16.973, -65.5, 103.517, -37.255, 17.666, 49.275]
  MoveL 1355 to (-1170, 550, -0.5) mm, rotated rx -180 ry 0 rz 90 deg; joints [16.973, -63.781, 104.061, -42.041, 15.922, 54.273]
  MoveL 1356 to (-1170, 550, 50) mm, rotated rx -180 ry 0 rz 90 deg; joints [16.973, -65.5, 103.517, -37.255, 17.666, 49.275]
  MoveL 1357 to (-1170, 600, 50) mm, rotated rx 180 ry 0 rz 90 deg; joints [17.465, -67.393, 106.361, -39.801, 17.161, 52.263]
  MoveL 1358 to (-1170, 600, -0.5) mm, rotated rx 180 ry 0 rz 90 deg; joints [17.465, -65.613, 106.914, -45.19, 15.44, 57.877]
  MoveL 1359 to (-1170, 600, 50) mm, rotated rx 180 ry 0 rz 90 deg; joints [17.465, -67.393, 106.361, -39.801, 17.161, 52.263]
  MoveL 1360 to (-1170, 650, 50) mm, rotated rx -180 ry 0 rz 90 deg; joints [17.986, -69.284, 109.144, -42.385, 16.754, 55.311]
  MoveL 1361 to (-1170, 650, -0.5) mm, rotated rx -180 ry 0 rz 90 deg; joints [17.986, -67.441, 109.706, -48.398, 15.062, 61.562]
  MoveL 1362 to (-1170, 650, 50) mm, rotated rx -180 ry 0 rz 90 deg; joints [17.986, -69.284, 109.144, -42.385, 16.754, 55.311]
  MoveL 1363 to (-1170, 700, 50) mm, rotated rx -180 ry 0 rz 90 deg; joints [18.537, -71.18, 111.869, -44.971, 16.445, 58.381]
  MoveL 1364 to (-1170, 700, -0.5) mm, rotated rx -180 ry 0 rz 90 deg; joints [18.537, -69.269, 112.442, -51.612, 14.789, 65.275]
  MoveL 1365 to (-1170, 700, 50) mm, rotated rx -180 ry 0 rz 90 deg; joints [18.537, -71.18, 111.869, -44.971, 16.445, 58.381]
  MoveL 1366 to (-1170, 750, 50) mm, rotated rx 180 ry 0 rz 90 deg; joints [19.122, -73.084, 114.539, -47.514, 16.234, 61.431]
  MoveL 1367 to (-1170, 750, -0.5) mm, rotated rx 180 ry 0 rz 90 deg; joints [19.122, -71.102, 115.125, -54.769, 14.619, 68.956]
  MoveL 1368 to (-1170, 750, 50) mm, rotated rx 180 ry 0 rz 90 deg; joints [19.122, -73.084, 114.539, -47.514, 16.234, 61.431]
  MoveL 1369 to (-1170, 800, 50) mm, rotated rx 180 ry 0 rz 90 deg; joints [19.744, -75.002, 117.156, -49.965, 16.121, 64.415]
  MoveL 1370 to (-1170, 800, -0.5) mm, rotated rx 180 ry 0 rz 90 deg; joints [19.744, -72.944, 117.757, -57.806, 14.55, 72.543]
  MoveL 1371 to (-1170, 800, 50) mm, rotated rx 180 ry 0 rz 90 deg; joints [19.744, -75.002, 117.156, -49.965, 16.121, 64.415]
  MoveL 1372 to (-1170, 850, 50) mm, rotated rx 180 ry 0 rz 90 deg; joints [20.406, -76.94, 119.723, -52.276, 16.106, 67.285]
  MoveL 1373 to (-1170, 850, -0.5) mm, rotated rx 180 ry 0 rz 90 deg; joints [20.406, -74.801, 120.341, -60.657, 14.579, 75.974]
  MoveL 1374 to (-1170, 850, 50) mm, rotated rx 180 ry 0 rz 90 deg; joints [20.406, -76.94, 119.723, -52.276, 16.106, 67.285]
  MoveL 1375 to (-1170, 900, 50) mm, rotated rx -180 ry 0 rz 90 deg; joints [21.111, -78.902, 122.242, -54.399, 16.187, 69.997]
  MoveL 1376 to (-1170, 900, -0.5) mm, rotated rx -180 ry 0 rz 90 deg; joints [21.111, -76.678, 122.877, -63.263, 14.703, 79.191]
  MoveL 1377 to (-1170, 900, 50) mm, rotated rx -180 ry 0 rz 90 deg; joints [21.111, -78.902, 122.242, -54.399, 16.187, 69.997]
  MoveL 1378 to (-1170, 950, 50) mm, rotated rx 180 ry 0 rz 90 deg; joints [21.864, -80.895, 124.713, -56.29, 16.364, 72.507]
  MoveL 1379 to (-1170, 950, -0.5) mm, rotated rx -180 ry 0 rz 90 deg; joints [21.864, -78.581, 125.368, -65.572, 14.916, 82.144]
  MoveL 1380 to (-1170, 950, 50) mm, rotated rx 180 ry 0 rz 90 deg; joints [21.864, -80.895, 124.713, -56.29, 16.364, 72.507]
  MoveL 1381 to (-1170, 1000, 50) mm, rotated rx 180 ry 0 rz 90 deg; joints [22.671, -82.925, 127.137, -57.909, 16.637, 74.78]
  MoveL 1382 to (-1170, 1000, -0.5) mm, rotated rx 180 ry 0 rz 90 deg; joints [22.671, -80.515, 127.814, -67.54, 15.217, 84.793]
  MoveL 1383 to (-1170, 1000, 50) mm, rotated rx 180 ry 0 rz 90 deg; joints [22.671, -82.925, 127.137, -57.909, 16.637, 74.78]
  MoveL 1384 to (-1170, 1050, 50) mm, rotated rx 180 ry 0 rz 90 deg; joints [23.535, -84.999, 129.514, -59.224, 17.007, 76.786]
  MoveL 1385 to (-1170, 1050, -0.5) mm, rotated rx 180 ry 0 rz 90 deg; joints [23.535, -82.487, 130.216, -69.133, 15.601, 87.107]
  MoveL 1386 to (-1170, 1050, 50) mm, rotated rx 180 ry 0 rz 90 deg; joints [23.535, -84.999, 129.514, -59.224, 17.007, 76.786]
  MoveL 1387 to (-1170, 1100, 50) mm, rotated rx 180 ry 0 rz 90 deg; joints [24.464, -87.126, 131.844, -60.213, 17.475, 78.504]
  MoveL 1388 to (-1170, 1100, -0.5) mm, rotated rx 180 ry 0 rz 90 deg; joints [24.464, -84.505, 132.574, -70.328, 16.068, 89.065]
  MoveL 1389 to (-1170, 1100, 50) mm, rotated rx 180 ry 0 rz 90 deg; joints [24.464, -87.126, 131.844, -60.213, 17.475, 78.504]
  MoveL 1390 to (-1170, 1150, 50) mm, rotated rx 180 ry 0 rz 90 deg; joints [25.465, -89.314, 134.126, -60.857, 18.047, 79.92]
  MoveL 1391 to (-1170, 1150, -0.5) mm, rotated rx -180 ry 0 rz 90 deg; joints [25.465, -86.577, 134.886, -71.108, 16.618, 90.655]
  MoveL 1392 to (-1170, 1150, 50) mm, rotated rx 180 ry 0 rz 90 deg; joints [25.465, -89.314, 134.126, -60.857, 18.047, 79.92]
  MoveL 1393 to (-1170, 1200, 50) mm, rotated rx 180 ry 0 rz 90 deg; joints [26.544, -91.571, 136.36, -61.149, 18.729, 81.03]
  MoveL 1394 to (-1170, 1200, -0.5) mm, rotated rx -180 ry 0 rz 90 deg; joints [26.544, -88.712, 137.153, -71.466, 17.255, 91.873]
  MoveL 1395 to (-1170, 1200, 50) mm, rotated rx 180 ry 0 rz 90 deg; joints [26.544, -91.571, 136.36, -61.149, 18.729, 81.03]
  MoveL 1396 to (-1170, 1250, 50) mm, rotated rx -180 ry 0 rz 90 deg; joints [27.711, -93.91, 138.542, -61.089, 19.531, 81.835]
  MoveL 1397 to (-1170, 1250, -0.5) mm, rotated rx -180 ry 0 rz 90 deg; joints [27.711, -90.921, 139.373, -71.4, 17.985, 92.721]
  MoveL 1398 to (-1170, 1250, 50) mm, rotated rx -180 ry 0 rz 90 deg; joints [27.711, -93.91, 138.542, -61.089, 19.531, 81.835]
  MoveL 1399 to (-1170, 1300, 50) mm, rotated rx -180 ry 0 rz 90 deg; joints [28.977, -96.341, 140.671, -60.685, 20.466, 82.349]
  MoveL 1400 to (-1170, 1300, -0.5) mm, rotated rx 180 ry 0 rz 90 deg; joints [28.977, -93.215, 141.542, -70.917, 18.821, 93.208]
  MoveL 1401 to (-1170, 1300, 50) mm, rotated rx -180 ry 0 rz 90 deg; joints [28.977, -96.341, 140.671, -60.685, 20.466, 82.349]
  MoveL 1402 to (-1170, 1350, 50) mm, rotated rx 180 ry 0 rz 90 deg; joints [30.352, -98.876, 142.744, -59.953, 21.554, 82.59]
  MoveL 1403 to (-1170, 1350, -0.5) mm, rotated rx -180 ry 0 rz 90 deg; joints [30.352, -95.608, 143.66, -70.027, 19.777, 93.351]
  MoveL 1404 to (-1170, 1350, 50) mm, rotated rx 180 ry 0 rz 90 deg; joints [30.352, -98.876, 142.744, -59.953, 21.554, 82.59]
  MoveL 1405 to (-1240, 50, 50) mm, rotated rx -180 ry 0 rz 90 deg; joints [14.958, -44.504, 68.794, -19.518, 29.089, 28.941]
  MoveL 1406 to (-1240, 50, -0.5) mm, rotated rx 180 ry 0 rz 90 deg; joints [14.958, -43.29, 69.348, -20.647, 27.43, 30.222]
  MoveL 1407 to (-1240, 50, 50) mm, rotated rx -180 ry 0 rz 90 deg; joints [14.958, -44.504, 68.794, -19.518, 29.089, 28.941]
  MoveL 1408 to (-1240, 100, 50) mm, rotated rx -180 ry 0 rz 90 deg; joints [15.294, -46.746, 72.724, -20.987, 27.612, 30.772]
  MoveL 1409 to (-1240, 100, -0.5) mm, rotated rx 180 ry 0 rz 90 deg; joints [15.294, -45.489, 73.266, -22.302, 25.94, 32.245]
  MoveL 1410 to (-1240, 100, 50) mm, rotated rx -180 ry 0 rz 90 deg; joints [15.294, -46.746, 72.724, -20.987, 27.612, 30.772]
  MoveL 1411 to (-1240, 150, 50) mm, rotated rx 180 ry 0 rz 90 deg; joints [15.646, -48.911, 76.476, -22.562, 26.254, 32.715]
  MoveL 1412 to (-1240, 150, -0.5) mm, rotated rx -180 ry 0 rz 90 deg; joints [15.646, -47.611, 77.01, -24.09, 24.57, 34.407]
  MoveL 1413 to (-1240, 150, 50) mm, rotated rx 180 ry 0 rz 90 deg; joints [15.646, -48.911, 76.476, -22.562, 26.254, 32.715]
  MoveL 1414 to (-1240, 200, 50) mm, rotated rx -180 ry 0 rz 90 deg; joints [16.013, -51.011, 80.075, -24.247, 25.007, 34.778]
  MoveL 1415 to (-1240, 200, -0.5) mm, rotated rx 180 ry 0 rz 90 deg; joints [16.013, -49.667, 80.603, -26.02, 23.312, 36.721]
  MoveL 1416 to (-1240, 200, 50) mm, rotated rx -180 ry 0 rz 90 deg; joints [16.013, -51.011, 80.075, -24.247, 25.007, 34.778]
  MoveL 1417 to (-1240, 250, 50) mm, rotated rx 180 ry 0 rz 90 deg; joints [16.398, -53.058, 83.54, -26.048, 23.865, 36.965]
  MoveL 1418 to (-1240, 250, -0.5) mm, rotated rx 180 ry 0 rz 90 deg; joints [16.398, -51.669, 84.065, -28.098, 22.161, 39.193]
  MoveL 1419 to (-1240, 250, 50) mm, rotated rx 180 ry 0 rz 90 deg; joints [16.398, -53.058, 83.54, -26.048, 23.865, 36.965]
  MoveL 1420 to (-1240, 300, 50) mm, rotated rx 180 ry 0 rz 90 deg; joints [16.801, -55.06, 86.886, -27.965, 22.824, 39.28]
  MoveL 1421 to (-1240, 300, -0.5) mm, rotated rx 180 ry 0 rz 90 deg; joints [16.801, -53.625, 87.409, -30.33, 21.114, 41.83]
  MoveL 1422 to (-1240, 300, 50) mm, rotated rx 180 ry 0 rz 90 deg; joints [16.801, -55.06, 86.886, -27.965, 22.824, 39.28]
  MoveL 1423 to (-1240, 350, 50) mm, rotated rx -180 ry 0 rz 90 deg; joints [17.224, -57.025, 90.125, -29.999, 21.882, 41.725]
  MoveL 1424 to (-1240, 350, -0.5) mm, rotated rx 180 ry 0 rz 90 deg; joints [17.224, -55.543, 90.649, -32.716, 20.168, 44.635]
  MoveL 1425 to (-1240, 350, 50) mm, rotated rx -180 ry 0 rz 90 deg; joints [17.224, -57.025, 90.125, -29.999, 21.882, 41.725]
  MoveL 1426 to (-1240, 400, 50) mm, rotated rx 180 ry 0 rz 90 deg; joints [17.668, -58.96, 93.269, -32.145, 21.037, 44.295]
  MoveL 1427 to (-1240, 400, -0.5) mm, rotated rx 180 ry 0 rz 90 deg; joints [17.668, -57.429, 93.795, -35.251, 19.325, 47.604]
  MoveL 1428 to (-1240, 400, 50) mm, rotated rx 180 ry 0 rz 90 deg; joints [17.668, -58.96, 93.269, -32.145, 21.037, 44.295]
  MoveL 1429 to (-1240, 450, 50) mm, rotated rx -180 ry 0 rz 90 deg; joints [18.134, -60.871, 96.326, -34.394, 20.289, 46.984]
  MoveL 1430 to (-1240, 450, -0.5) mm, rotated rx -180 ry 0 rz 90 deg; joints [18.134, -59.288, 96.855, -37.927, 18.582, 50.73]
  MoveL 1431 to (-1240, 450, 50) mm, rotated rx -180 ry 0 rz 90 deg; joints [18.134, -60.871, 96.326, -34.394, 20.289, 46.984]
  MoveL 1432 to (-1240, 500, 50) mm, rotated rx 180 ry 0 rz 90 deg; joints [18.625, -62.763, 99.303, -36.733, 19.637, 49.779]
  MoveL 1433 to (-1240, 500, -0.5) mm, rotated rx -180 ry 0 rz 90 deg; joints [18.625, -61.126, 99.837, -40.725, 17.942, 53.996]
  MoveL 1434 to (-1240, 500, 50) mm, rotated rx 180 ry 0 rz 90 deg; joints [18.625, -62.763, 99.303, -36.733, 19.637, 49.779]
  MoveL 1435 to (-1240, 550, 50) mm, rotated rx -180 ry 0 rz 90 deg; joints [19.142, -64.64, 102.206, -39.142, 19.082, 52.663]
  MoveL 1436 to (-1240, 550, -0.5) mm, rotated rx -180 ry 0 rz 90 deg; joints [19.142, -62.948, 102.746, -43.622, 17.405, 57.379]
  MoveL 1437 to (-1240, 550, 50) mm, rotated rx -180 ry 0 rz 90 deg; joints [19.142, -64.64, 102.206, -39.142, 19.082, 52.663]
  MoveL 1438 to (-1240, 600, 50) mm, rotated rx -180 ry 0 rz 90 deg; joints [19.688, -66.509, 105.04, -41.597, 18.624, 55.613]
  MoveL 1439 to (-1240, 600, -0.5) mm, rotated rx -180 ry 0 rz 90 deg; joints [19.688, -64.758, 105.588, -46.582, 16.971, 60.848]
  MoveL 1440 to (-1240, 600, 50) mm, rotated rx -180 ry 0 rz 90 deg; joints [19.688, -66.509, 105.04, -41.597, 18.624, 55.613]
  MoveL 1441 to (-1240, 650, 50) mm, rotated rx 180 ry 0 rz 90 deg; joints [20.264, -68.372, 107.81, -44.068, 18.264, 58.6]
  MoveL 1442 to (-1240, 650, -0.5) mm, rotated rx 180 ry 0 rz 90 deg; joints [20.264, -66.56, 108.367, -49.567, 16.64, 64.363]
  MoveL 1443 to (-1240, 650, 50) mm, rotated rx 180 ry 0 rz 90 deg; joints [20.264, -68.372, 107.81, -44.068, 18.264, 58.6]
  MoveL 1444 to (-1240, 700, 50) mm, rotated rx 180 ry 0 rz 90 deg; joints [20.874, -70.236, 110.52, -46.52, 18.001, 61.591]
  MoveL 1445 to (-1240, 700, -0.5) mm, rotated rx 180 ry 0 rz 90 deg; joints [20.874, -68.359, 111.088, -52.529, 16.411, 67.88]
  MoveL 1446 to (-1240, 700, 50) mm, rotated rx 180 ry 0 rz 90 deg; joints [20.874, -70.236, 110.52, -46.52, 18.001, 61.591]
  MoveL 1447 to (-1240, 750, 50) mm, rotated rx -180 ry 0 rz 90 deg; joints [21.52, -72.103, 113.172, -48.914, 17.835, 64.549]
  MoveL 1448 to (-1240, 750, -0.5) mm, rotated rx 180 ry 0 rz 90 deg; joints [21.52, -70.158, 113.752, -55.417, 16.284, 71.35]
  MoveL 1449 to (-1240, 750, 50) mm, rotated rx -180 ry 0 rz 90 deg; joints [21.52, -72.103, 113.172, -48.914, 17.835, 64.549]
  MoveL 1450 to (-1240, 800, 50) mm, rotated rx -180 ry 0 rz 90 deg; joints [22.204, -73.98, 115.77, -51.21, 17.765, 67.436]
  MoveL 1451 to (-1240, 800, -0.5) mm, rotated rx -180 ry 0 rz 90 deg; joints [22.204, -71.963, 116.363, -58.179, 16.254, 74.723]
  MoveL 1452 to (-1240, 800, 50) mm, rotated rx -180 ry 0 rz 90 deg; joints [22.204, -73.98, 115.77, -51.21, 17.765, 67.436]
  MoveL 1453 to (-1240, 850, 50) mm, rotated rx 180 ry 0 rz 90 deg; joints [22.932, -75.87, 118.315, -53.368, 17.792, 70.215]
  MoveL 1454 to (-1240, 850, -0.5) mm, rotated rx 180 ry 0 rz 90 deg; joints [22.932, -73.776, 118.923, -60.766, 16.32, 77.951]
  MoveL 1455 to (-1240, 850, 50) mm, rotated rx 180 ry 0 rz 90 deg; joints [22.932, -75.87, 118.315, -53.368, 17.792, 70.215]
  MoveL 1456 to (-1240, 900, 50) mm, rotated rx 180 ry 0 rz 90 deg; joints [23.705, -77.777, 120.809, -55.35, 17.912, 72.848]
  MoveL 1457 to (-1240, 900, -0.5) mm, rotated rx 180 ry 0 rz 90 deg; joints [23.705, -75.603, 121.433, -63.13, 16.477, 80.991]
  MoveL 1458 to (-1240, 900, 50) mm, rotated rx 180 ry 0 rz 90 deg; joints [23.705, -77.777, 120.809, -55.35, 17.912, 72.848]
  MoveL 1459 to (-1240, 950, 50) mm, rotated rx 180 ry 0 rz 90 deg; joints [24.53, -79.708, 123.252, -57.121, 18.126, 75.305]
  MoveL 1460 to (-1240, 950, -0.5) mm, rotated rx -180 ry 0 rz 90 deg; joints [24.53, -77.449, 123.896, -65.232, 16.723, 83.805]
  MoveL 1461 to (-1240, 950, 50) mm, rotated rx 180 ry 0 rz 90 deg; joints [24.53, -79.708, 123.252, -57.121, 18.126, 75.305]
  MoveL 1462 to (-1240, 1000, 50) mm, rotated rx 180 ry 0 rz 90 deg; joints [25.41, -81.667, 125.646, -58.65, 18.433, 77.556]
  MoveL 1463 to (-1240, 1000, -0.5) mm, rotated rx -180 ry 0 rz 90 deg; joints [25.41, -79.317, 126.31, -67.04, 17.054, 86.363]
  MoveL 1464 to (-1240, 1000, 50) mm, rotated rx 180 ry 0 rz 90 deg; joints [25.41, -81.667, 125.646, -58.65, 18.433, 77.556]
  MoveL 1465 to (-1240, 1050, 50) mm, rotated rx 180 ry 0 rz 90 deg; joints [26.35, -83.661, 127.991, -59.914, 18.834, 79.581]
  MoveL 1466 to (-1240, 1050, -0.5) mm, rotated rx 180 ry 0 rz 90 deg; joints [26.35, -81.215, 128.677, -68.527, 17.467, 88.644]
  MoveL 1467 to (-1240, 1050, 50) mm, rotated rx 180 ry 0 rz 90 deg; joints [26.35, -83.661, 127.991, -59.914, 18.834, 79.581]
  MoveL 1468 to (-1240, 1100, 50) mm, rotated rx 180 ry 0 rz 90 deg; joints [27.358, -85.694, 130.286, -60.893, 19.33, 81.365]
  MoveL 1469 to (-1240, 1100, -0.5) mm, rotated rx -180 ry 0 rz 90 deg; joints [27.358, -83.146, 130.998, -69.677, 17.963, 90.632]
  MoveL 1470 to (-1240, 1100, 50) mm, rotated rx 180 ry 0 rz 90 deg; joints [27.358, -85.694, 130.286, -60.893, 19.33, 81.365]
  MoveL 1471 to (-1240, 1150, 50) mm, rotated rx -180 ry 0 rz 90 deg; joints [28.439, -87.773, 132.531, -61.577, 19.924, 82.897]
  MoveL 1472 to (-1240, 1150, -0.5) mm, rotated rx -180 ry 0 rz 90 deg; joints [28.439, -85.119, 133.27, -70.476, 18.541, 92.32]
  MoveL 1473 to (-1240, 1150, 50) mm, rotated rx -180 ry 0 rz 90 deg; joints [28.439, -87.773, 132.531, -61.577, 19.924, 82.897]
  MoveL 1474 to (-1240, 1200, 50) mm, rotated rx -180 ry 0 rz 90 deg; joints [29.601, -89.907, 134.725, -61.958, 20.622, 84.177]
  MoveL 1475 to (-1240, 1200, -0.5) mm, rotated rx 180 ry 0 rz 90 deg; joints [29.601, -87.138, 135.493, -70.921, 19.204, 93.706]
  MoveL 1476 to (-1240, 1200, 50) mm, rotated rx -180 ry 0 rz 90 deg; joints [29.601, -89.907, 134.725, -61.958, 20.622, 84.177]
  MoveL 1477 to (-1240, 1250, 50) mm, rotated rx -180 ry 0 rz 90 deg; joints [30.852, -92.101, 136.865, -62.038, 21.431, 85.207]
  MoveL 1478 to (-1240, 1250, -0.5) mm, rotated rx 180 ry 0 rz 90 deg; joints [30.852, -89.212, 137.667, -71.01, 19.957, 94.794]
  MoveL 1479 to (-1240, 1250, 50) mm, rotated rx -180 ry 0 rz 90 deg; joints [30.852, -92.101, 136.865, -62.038, 21.431, 85.207]
  MoveL 1480 to (-1240, 1300, 50) mm, rotated rx 180 ry 0 rz 90 deg; joints [32.202, -94.363, 138.95, -61.822, 22.362, 85.997]
  MoveL 1481 to (-1240, 1300, -0.5) mm, rotated rx 180 ry 0 rz 90 deg; joints [32.202, -91.348, 139.787, -70.75, 20.808, 95.594]
  MoveL 1482 to (-1240, 1300, 50) mm, rotated rx 180 ry 0 rz 90 deg; joints [32.202, -94.363, 138.95, -61.822, 22.362, 85.997]
  MoveL 1483 to (-1240, 1350, 50) mm, rotated rx -180 ry 0 rz 90 deg; joints [33.661, -96.702, 140.975, -61.323, 23.428, 86.564]
  MoveL 1484 to (-1240, 1350, -0.5) mm, rotated rx 180 ry 0 rz 90 deg; joints [33.661, -93.555, 141.853, -70.149, 21.769, 96.12]
  MoveL 1485 to (-1240, 1350, 50) mm, rotated rx -180 ry 0 rz 90 deg; joints [33.661, -96.702, 140.975, -61.323, 23.428, 86.564]
  MoveL 1486 to (-1240, 1400, 50) mm, rotated rx 180 ry 0 rz 90 deg; joints [35.241, -99.125, 142.938, -60.561, 24.644, 86.932]
  MoveL 1487 to (-1240, 1400, -0.5) mm, rotated rx 180 ry 0 rz 90 deg; joints [35.241, -95.842, 143.859, -69.224, 22.854, 96.392]
  MoveL 1488 to (-1240, 1400, 50) mm, rotated rx 180 ry 0 rz 90 deg; joints [35.241, -99.125, 142.938, -60.561, 24.644, 86.932]
  MoveL 1489 to (-1240, 1450, 50) mm, rotated rx 180 ry 0 rz 90 deg; joints [36.955, -101.64, 144.834, -59.558, 26.03, 87.128]
  MoveL 1490 to (-1240, 1450, -0.5) mm, rotated rx -180 ry 0 rz 90 deg; joints [36.955, -98.216, 145.803, -67.998, 24.083, 96.44]
  MoveL 1491 to (-1240, 1450, 50) mm, rotated rx 180 ry 0 rz 90 deg; joints [36.955, -101.64, 144.834, -59.558, 26.03, 87.128]
  MoveL 1492 to (-1310, 50, 50) mm, rotated rx 180 ry 0 rz 90 deg; joints [16.668, -43.593, 67.188, -20.974, 30.284, 31.415]
  MoveL 1493 to (-1310, 50, -0.5) mm, rotated rx 180 ry 0 rz 90 deg; joints [16.668, -42.397, 67.747, -22.115, 28.651, 32.725]
  MoveL 1494 to (-1310, 50, 50) mm, rotated rx 180 ry 0 rz 90 deg; joints [16.668, -43.593, 67.188, -20.974, 30.284, 31.415]
  MoveL 1495 to (-1310, 100, 50) mm, rotated rx -180 ry 0 rz 90 deg; joints [17.039, -45.85, 71.159, -22.494, 28.816, 33.338]
  MoveL 1496 to (-1310, 100, -0.5) mm, rotated rx -180 ry 0 rz 90 deg; joints [17.039, -44.611, 71.706, -23.814, 27.174, 34.833]
  MoveL 1497 to (-1310, 100, 50) mm, rotated rx -180 ry 0 rz 90 deg; joints [17.039, -45.85, 71.159, -22.494, 28.816, 33.338]
  MoveL 1498 to (-1310, 150, 50) mm, rotated rx 180 ry 0 rz 90 deg; joints [17.425, -48.024, 74.944, -24.111, 27.473, 35.365]
  MoveL 1499 to (-1310, 150, -0.5) mm, rotated rx -180 ry 0 rz 90 deg; joints [17.425, -46.742, 75.481, -25.636, 25.823, 37.071]
  MoveL 1500 to (-1310, 150, 50) mm, rotated rx 180 ry 0 rz 90 deg; joints [17.425, -48.024, 74.944, -24.111, 27.473, 35.365]
  MoveL 1501 to (-1310, 200, 50) mm, rotated rx 180 ry 0 rz 90 deg; joints [17.829, -50.128, 78.567, -25.83, 26.247, 37.502]
  MoveL 1502 to (-1310, 200, -0.5) mm, rotated rx 180 ry 0 rz 90 deg; joints [17.829, -48.803, 79.097, -27.585, 24.59, 39.445]
  MoveL 1503 to (-1310, 200, 50) mm, rotated rx 180 ry 0 rz 90 deg; joints [17.829, -50.128, 78.567, -25.83, 26.247, 37.502]
  MoveL 1504 to (-1310, 250, 50) mm, rotated rx -180 ry 0 rz 90 deg; joints [18.252, -52.175, 82.05, -27.653, 25.131, 39.753]
  MoveL 1505 to (-1310, 250, -0.5) mm, rotated rx 180 ry 0 rz 90 deg; joints [18.252, -50.806, 82.576, -29.667, 23.467, 41.962]
  MoveL 1506 to (-1310, 250, 50) mm, rotated rx -180 ry 0 rz 90 deg; joints [18.252, -52.175, 82.05, -27.653, 25.131, 39.753]
  MoveL 1507 to (-1310, 300, 50) mm, rotated rx -180 ry 0 rz 90 deg; joints [18.695, -54.173, 85.408, -29.579, 24.119, 42.12]
  MoveL 1508 to (-1310, 300, -0.5) mm, rotated rx -180 ry 0 rz 90 deg; joints [18.695, -52.759, 85.932, -31.881, 22.453, 44.625]
  MoveL 1509 to (-1310, 300, 50) mm, rotated rx -180 ry 0 rz 90 deg; joints [18.695, -54.173, 85.408, -29.579, 24.119, 42.12]
  MoveL 1510 to (-1310, 350, 50) mm, rotated rx 180 ry 0 rz 90 deg; joints [19.158, -56.131, 88.656, -31.606, 23.209, 44.6]
  MoveL 1511 to (-1310, 350, -0.5) mm, rotated rx -180 ry 0 rz 90 deg; joints [19.158, -54.67, 89.18, -34.225, 21.543, 47.432]
  MoveL 1512 to (-1310, 350, 50) mm, rotated rx 180 ry 0 rz 90 deg; joints [19.158, -56.131, 88.656, -31.606, 23.209, 44.6]
  MoveL 1513 to (-1310, 400, 50) mm, rotated rx 180 ry 0 rz 90 deg; joints [19.644, -58.055, 91.804, -33.727, 22.398, 47.188]
  MoveL 1514 to (-1310, 400, -0.5) mm, rotated rx 180 ry 0 rz 90 deg; joints [19.644, -56.547, 92.328, -36.693, 20.737, 50.377]
  MoveL 1515 to (-1310, 400, 50) mm, rotated rx 180 ry 0 rz 90 deg; joints [19.644, -58.055, 91.804, -33.727, 22.398, 47.188]
  MoveL 1516 to (-1310, 450, 50) mm, rotated rx 180 ry 0 rz 90 deg; joints [20.155, -59.951, 94.86, -35.931, 21.686, 49.877]
  MoveL 1517 to (-1310, 450, -0.5) mm, rotated rx -180 ry 0 rz 90 deg; joints [20.155, -58.393, 95.388, -39.27, 20.033, 53.45]
  MoveL 1518 to (-1310, 450, 50) mm, rotated rx 180 ry 0 rz 90 deg; joints [20.155, -59.951, 94.86, -35.931, 21.686, 49.877]
  MoveL 1519 to (-1310, 500, 50) mm, rotated rx -180 ry 0 rz 90 deg; joints [20.692, -61.825, 97.833, -38.203, 21.072, 52.651]
  MoveL 1520 to (-1310, 500, -0.5) mm, rotated rx 180 ry 0 rz 90 deg; joints [20.692, -60.216, 98.365, -41.94, 19.433, 56.634]
  MoveL 1521 to (-1310, 500, 50) mm, rotated rx -180 ry 0 rz 90 deg; joints [20.692, -61.825, 97.833, -38.203, 21.072, 52.651]
  MoveL 1522 to (-1310, 550, 50) mm, rotated rx 180 ry 0 rz 90 deg; joints [21.256, -63.681, 100.73, -40.525, 20.556, 55.495]
  MoveL 1523 to (-1310, 550, -0.5) mm, rotated rx -180 ry 0 rz 90 deg; joints [21.256, -62.018, 101.267, -44.676, 18.935, 59.904]
  MoveL 1524 to (-1310, 550, 50) mm, rotated rx 180 ry 0 rz 90 deg; joints [21.256, -63.681, 100.73, -40.525, 20.556, 55.495]
  MoveL 1525 to (-1310, 600, 50) mm, rotated rx 180 ry 0 rz 90 deg; joints [21.851, -65.525, 103.555, -42.873, 20.137, 58.385]
  MoveL 1526 to (-1310, 600, -0.5) mm, rotated rx -180 ry 0 rz 90 deg; joints [21.851, -63.805, 104.099, -47.448, 18.539, 63.233]
  MoveL 1527 to (-1310, 600, 50) mm, rotated rx 180 ry 0 rz 90 deg; joints [21.851, -65.525, 103.555, -42.873, 20.137, 58.385]
  MoveL 1528 to (-1310, 650, 50) mm, rotated rx -180 ry 0 rz 90 deg; joints [22.478, -67.36, 106.313, -45.219, 19.815, 61.297]
  MoveL 1529 to (-1310, 650, -0.5) mm, rotated rx 180 ry 0 rz 90 deg; joints [22.478, -65.581, 106.865, -50.22, 18.245, 66.587]
  MoveL 1530 to (-1310, 650, 50) mm, rotated rx -180 ry 0 rz 90 deg; joints [22.478, -67.36, 106.313, -45.219, 19.815, 61.297]
  MoveL 1531 to (-1310, 700, 50) mm, rotated rx 180 ry 0 rz 90 deg; joints [23.14, -69.19, 109.007, -47.532, 19.589, 64.2]
  MoveL 1532 to (-1310, 700, -0.5) mm, rotated rx 180 ry 0 rz 90 deg; joints [23.14, -67.35, 109.569, -52.953, 18.051, 69.926]
  MoveL 1533 to (-1310, 700, 50) mm, rotated rx 180 ry 0 rz 90 deg; joints [23.14, -69.19, 109.007, -47.532, 19.589, 64.2]
  MoveL 1534 to (-1310, 750, 50) mm, rotated rx 180 ry 0 rz 90 deg; joints [23.84, -71.02, 111.642, -49.78, 19.459, 67.065]
  MoveL 1535 to (-1310, 750, -0.5) mm, rotated rx 180 ry 0 rz 90 deg; joints [23.84, -69.115, 112.214, -55.604, 17.955, 73.212]
  MoveL 1536 to (-1310, 750, 50) mm, rotated rx 180 ry 0 rz 90 deg; joints [23.84, -71.02, 111.642, -49.78, 19.459, 67.065]
  MoveL 1537 to (-1310, 800, 50) mm, rotated rx 180 ry 0 rz 90 deg; joints [24.581, -72.853, 114.219, -51.929, 19.423, 69.859]
  MoveL 1538 to (-1310, 800, -0.5) mm, rotated rx 180 ry 0 rz 90 deg; joints [24.581, -70.88, 114.804, -58.131, 17.954, 76.405]
  MoveL 1539 to (-1310, 800, 50) mm, rotated rx 180 ry 0 rz 90 deg; joints [24.581, -72.853, 114.219, -51.929, 19.423, 69.859]
  MoveL 1540 to (-1310, 850, 50) mm, rotated rx 180 ry 0 rz 90 deg; joints [25.367, -74.694, 116.741, -53.946, 19.48, 72.552]
  MoveL 1541 to (-1310, 850, -0.5) mm, rotated rx 180 ry 0 rz 90 deg; joints [25.367, -72.648, 117.339, -60.495, 18.046, 79.468]
  MoveL 1542 to (-1310, 850, 50) mm, rotated rx 180 ry 0 rz 90 deg; joints [25.367, -74.694, 116.741, -53.946, 19.48, 72.552]
  MoveL 1543 to (-1310, 900, 50) mm, rotated rx 180 ry 0 rz 90 deg; joints [26.201, -76.546, 119.209, -55.8, 19.63, 75.116]
  MoveL 1544 to (-1310, 900, -0.5) mm, rotated rx -180 ry 0 rz 90 deg; joints [26.201, -74.425, 119.823, -62.66, 18.228, 82.366]
  MoveL 1545 to (-1310, 900, 50) mm, rotated rx 180 ry 0 rz 90 deg; joints [26.201, -76.546, 119.209, -55.8, 19.63, 75.116]
  MoveL 1546 to (-1310, 950, 50) mm, rotated rx 180 ry 0 rz 90 deg; joints [27.087, -78.414, 121.624, -57.464, 19.871, 77.525]
  MoveL 1547 to (-1310, 950, -0.5) mm, rotated rx 180 ry 0 rz 90 deg; joints [27.087, -76.212, 122.255, -64.593, 18.496, 85.071]
  MoveL 1548 to (-1310, 950, 50) mm, rotated rx 180 ry 0 rz 90 deg; joints [27.087, -78.414, 121.624, -57.464, 19.871, 77.525]
  MoveL 1549 to (-1310, 1000, 50) mm, rotated rx 180 ry 0 rz 90 deg; joints [28.03, -80.302, 123.987, -58.913, 20.202, 79.758]
  MoveL 1550 to (-1310, 1000, -0.5) mm, rotated rx 180 ry 0 rz 90 deg; joints [28.03, -78.015, 124.636, -66.27, 18.848, 87.561]
  MoveL 1551 to (-1310, 1000, 50) mm, rotated rx 180 ry 0 rz 90 deg; joints [28.03, -80.302, 123.987, -58.913, 20.202, 79.758]
  MoveL 1552 to (-1310, 1050, 50) mm, rotated rx 180 ry 0 rz 90 deg; joints [29.035, -82.214, 126.298, -60.129, 20.624, 81.799]
  MoveL 1553 to (-1310, 1050, -0.5) mm, rotated rx 180 ry 0 rz 90 deg; joints [29.035, -79.838, 126.968, -67.67, 19.281, 89.819]
  MoveL 1554 to (-1310, 1050, 50) mm, rotated rx 180 ry 0 rz 90 deg; joints [29.035, -82.214, 126.298, -60.129, 20.624, 81.799]
  MoveL 1555 to (-1310, 1100, 50) mm, rotated rx 180 ry 0 rz 90 deg; joints [30.108, -84.154, 128.557, -61.097, 21.137, 83.636]
  MoveL 1556 to (-1310, 1100, -0.5) mm, rotated rx -180 ry 0 rz 90 deg; joints [30.108, -81.684, 129.249, -68.78, 19.795, 91.835]
  MoveL 1557 to (-1310, 1100, 50) mm, rotated rx 180 ry 0 rz 90 deg; joints [30.108, -84.154, 128.557, -61.097, 21.137, 83.636]
  MoveL 1558 to (-1310, 1150, 50) mm, rotated rx 180 ry 0 rz 90 deg; joints [31.255, -86.128, 130.763, -61.808, 21.745, 85.264]
  MoveL 1559 to (-1310, 1150, -0.5) mm, rotated rx -180 ry 0 rz 90 deg; joints [31.255, -83.558, 131.48, -69.592, 20.389, 93.603]
  MoveL 1560 to (-1310, 1150, 50) mm, rotated rx 180 ry 0 rz 90 deg; joints [31.255, -86.128, 130.763, -61.808, 21.745, 85.264]
